// 7.1 Контроль доступа (СКУД)
fbAccessControl(
    VI_System_Time_MS := GVL_STATUS.G_System_Time_MS,
    VI_IsActivePLC := GVL_STATUS.G_Is_Active_PLC,
    VI_Armed := GVL_ALARM.G_Security_Armed,
    VI_System_Mode := GVL_STATE.G_System_Mode,
    VI_Gate_Open_Req := GVL_CONFIG.G_HMI_Gate_Open_Req,
    VI_Wicket_Open_Req := GVL_CONFIG.G_HMI_Wicket_Open_Req,
    VI_Lock_1_Open_Req := GVL_CONFIG.G_HMI_Lock_1_Open_Req,
    VI_Lock_1_Close_Req := GVL_CONFIG.G_HMI_Lock_1_Close_Req,
    VI_Lock_2_Open_Req := GVL_CONFIG.G_HMI_Lock_2_Open_Req,
    VI_Lock_2_Close_Req := GVL_CONFIG.G_HMI_Lock_2_Close_Req,
    VI_PIN_Code := GVL_INTENT_USER.I_PIN_Code,
    VI_RFID_Tag := GVL_INTENT_USER.I_RFID_Tag,
    VI_Access_Codes := GVL_Retain.G_Access_Codes,
    VI_RFID_Tags := GVL_Retain.G_RFID_Tags,
    VI_Config := GVL_CONFIG.G_Security_Config,
    VO_Gate_Open => GVL_INTENT_USER.I_Gate_Open_Request,
    VO_Wicket_Open => GVL_INTENT_USER.I_Wicket_Open_Request,
    VO_Lock_1_Open => GVL_INTENT_USER.I_Lock_1_Open_Request,
    VO_Lock_1_Close => GVL_INTENT_USER.I_Lock_1_Close_Request,
    VO_Lock_2_Open => GVL_INTENT_USER.I_Lock_2_Open_Request,
    VO_Lock_2_Close => GVL_INTENT_USER.I_Lock_2_Close_Request
);
          
END_PROGRAM

PROGRAM PRG_Safety_Operator
  VAR
    fbSafetyWorkflow : FB_Safety_Workflow_Manager;
  END_VAR

            // Operator / test / recover workflow ownership.

fbSafetyWorkflow(
    VI_System_Time_MS := GVL_TIME_SERVICE.G_Now_MS,
    VI_Water_Selective_Recover := GVL_INTENT_USER.I_Water_Selective_Recover,
    VI_Gas_Selective_Recover := GVL_INTENT_USER.I_Gas_Selective_Recover,
    VI_Water_Valve_Test_Open := GVL_INTENT_USER.I_Water_Valve_Test_Open,
    VI_Water_Valve_Test_Close := GVL_INTENT_USER.I_Water_Valve_Test_Close,
    VI_Water_Valve_Test_Confirm := GVL_INTENT_USER.I_Water_Valve_Test_Confirm,
    VI_Gas_Valve_Test_Open := GVL_INTENT_USER.I_Gas_Valve_Test_Open,
    VI_Gas_Valve_Test_Close := GVL_INTENT_USER.I_Gas_Valve_Test_Close,
    VI_Gas_Valve_Test_Confirm := GVL_INTENT_USER.I_Gas_Valve_Test_Confirm
);

// propagate test timeout safety actions
IF fbSafetyWorkflow.VO_Water_Test_Timeout_Close_Required THEN
    GVL_INTENT_SAFETY.I_Test_Timeout_Water_Close := TRUE;
END_IF;

IF fbSafetyWorkflow.VO_Gas_Test_Timeout_Close_Required THEN
    GVL_INTENT_SAFETY.I_Test_Timeout_Gas_Close := TRUE;
END_IF;

// move recovery manual confirm here
IF GVL_INTENT_USER.I_Reset_Errors THEN
    GVL_SAFETY_RECOVERY.G_Recovery_Manual_Confirm := TRUE;
END_IF;

// >>> BULK_SYNC_ANCHOR: PRG_Safety_Operator <<<
          
END_PROGRAM

PROGRAM PRG_System_Runtime_Base
  VAR
    fbSystemInit : FB_System_Init;
    fbSystemRecovery : FB_System_Recovery;
    fbSystemPersist : FB_System_Persist_Manager;
    L_Local_State : ST_System_State_Snapshot;
    L_Remote_State : ST_System_State_Snapshot;
    L_Persist_Buffer : ARRAY[0..4] OF BYTE;
    L_Last_Written_Persist_Buffer : ARRAY[0..4] OF BYTE;
    L_Persist_Buffer_Changed : BOOL;
    L_Last_Persist_Write_MS : UDINT;
    L_Recovery_Done : BOOL;
    L_NVRAM_Cmd : BYTE;
    L_NVRAM_Offset : UDINT;
    L_NVRAM_Done : BOOL;
    L_NVRAM_Err : BOOL;
    L_NVRAM_ErrID : UDINT;
  END_VAR

            // ======================================================
// SYSTEM RUNTIME BASE
// ======================================================
// Initializes and maintains base system runtime helpers.
//
// Legacy direct-state redundancy orchestration is intentionally
// disconnected from active runtime execution.
// Current HA/distributed runtime path is:
// PRG_Peer_Heartbeat_Ingestion -> PRG_Peer_Session_Publication
// -> PRG_HA_Session_Replication -> distributed ingestion/governors.
//
// Do not reconnect FB_System_Redundancy_Orchestrator here without
// explicit barrier/governance review.
// ======================================================

fbSystemInit(
    VIO_Local_State := L_Local_State,
    VIO_Remote_State := L_Remote_State
);

fbSystemRecovery(
    VIO_Recovery_Done := L_Recovery_Done
);

fbSystemPersist(
    VI_System_Time_MS := GVL_TIME_SERVICE.G_Now_MS,
    VI_IsActivePLC := GVL_STATUS.G_Is_Active_PLC,
    VIO_Persist_Buffer := L_Persist_Buffer,
    VIO_Last_Written_Persist_Buffer := L_Last_Written_Persist_Buffer,
    VIO_Persist_Buffer_Changed := L_Persist_Buffer_Changed,
    VIO_Last_Persist_Write_MS := L_Last_Persist_Write_MS,
    VIO_NVRAM_Cmd := L_NVRAM_Cmd,
    VIO_NVRAM_Offset := L_NVRAM_Offset,
    VIO_NVRAM_Done := L_NVRAM_Done,
    VIO_NVRAM_Err := L_NVRAM_Err,
    VIO_NVRAM_ErrID := L_NVRAM_ErrID
);

// >>> BULK_SYNC_ANCHOR: PRG_System_Runtime_Base <<<
          
END_PROGRAM

PROGRAM PRG_Distributed_Snapshot_Governor
  VAR
    L_Now_MS : UDINT;
    L_Delta_MS : UDINT;
    L_Distributed_Snapshot_Valid : BOOL := TRUE;
    L_Error_Code : UDINT := 0;
    L_Error_Text : STRING(160) := '';
    L_Peer_Session_Active : BOOL := FALSE;
  END_VAR

            L_Now_MS := GVL_STATUS.G_System_Time_MS;
L_Distributed_Snapshot_Valid := TRUE;
L_Error_Code := 0;
L_Error_Text := '';

// ======================================================
// DISTRIBUTED IMMUTABLE SNAPSHOT GOVERNOR
// ======================================================
// Governs immutable peer publication snapshot exchange.
// Publication-authoritative only.
// Does not invalidate runtime barrier, PLC fencing
// or local immutable snapshot freeze.
//
// Recovery/release is convergence-lease based:
// distributed snapshot quarantine is not released on a
// single healthy scan.
// ======================================================

GVL_DISTRIBUTED_SNAPSHOT.Peer_Publication_Stale := FALSE;
GVL_DISTRIBUTED_SNAPSHOT.Peer_Snapshot_Not_Immutable := FALSE;
GVL_DISTRIBUTED_SNAPSHOT.Peer_Publication_Divergence := FALSE;
GVL_DISTRIBUTED_SNAPSHOT.Peer_Publication_Reconciliation_Lost := FALSE;
GVL_DISTRIBUTED_SNAPSHOT.Peer_Snapshot_Lease_Expired := FALSE;

// ------------------------------------------------------
// Local immutable publication projection.
// ------------------------------------------------------
// Distributed snapshot is upstream of output freshness in MAIN.
// Therefore local publication baseline must not read GVL_OUTPUT_EPOCH.
// It uses the already-frozen runtime snapshot epoch instead.
// ------------------------------------------------------

GVL_DISTRIBUTED_SNAPSHOT.Local_Distributed_Snapshot_Epoch := GVL_DISTRIBUTED_SNAPSHOT.Distributed_Snapshot_Epoch;
GVL_DISTRIBUTED_SNAPSHOT.Local_Runtime_Snapshot_Epoch := GVL_RUNTIME_SNAPSHOT.Snapshot_Epoch;
GVL_DISTRIBUTED_SNAPSHOT.Local_Publication_Epoch := GVL_RUNTIME_SNAPSHOT.Snapshot_Publication_Epoch;

// ------------------------------------------------------
// Local immutable publication freeze semantics.
// ------------------------------------------------------

IF GVL_RUNTIME_SNAPSHOT.Snapshot_Frozen
AND GVL_RUNTIME_SNAPSHOT.Snapshot_Publication_Allowed
AND GVL_RUNTIME_SNAPSHOT.Snapshot_Copy_Valid
AND GVL_RUNTIME_SNAPSHOT.Snapshot_Isolation_Valid
THEN
    GVL_DISTRIBUTED_SNAPSHOT.Distributed_Snapshot_Frozen := TRUE;
ELSE
    GVL_DISTRIBUTED_SNAPSHOT.Distributed_Snapshot_Frozen := FALSE;

    L_Distributed_Snapshot_Valid := FALSE;
    L_Error_Code := 14000;
    L_Error_Text := 'Local immutable snapshot not frozen';
END_IF;

// ------------------------------------------------------
// Peer session detection.
// ------------------------------------------------------

IF GVL_DISTRIBUTED_SNAPSHOT.Peer_Publication_Epoch > 0 THEN
    L_Peer_Session_Active := TRUE;
END_IF;

IF GVL_DISTRIBUTED_SNAPSHOT.Peer_Runtime_Snapshot_Epoch > 0 THEN
    L_Peer_Session_Active := TRUE;
END_IF;

IF GVL_DISTRIBUTED_SNAPSHOT.Peer_Distributed_Snapshot_Epoch > 0 THEN
    L_Peer_Session_Active := TRUE;
END_IF;

IF GVL_DISTRIBUTED_SNAPSHOT.Peer_Snapshot_Immutable THEN
    L_Peer_Session_Active := TRUE;
END_IF;

// ------------------------------------------------------
// Peer snapshot lease validation.
// ------------------------------------------------------

IF L_Distributed_Snapshot_Valid AND L_Peer_Session_Active THEN
    L_Delta_MS := L_Now_MS - GVL_DISTRIBUTED_SNAPSHOT.Peer_Snapshot_Last_Refresh_MS;

    IF GVL_DISTRIBUTED_SNAPSHOT.Peer_Snapshot_Lease_Active THEN
        IF L_Delta_MS > GVL_DISTRIBUTED_SNAPSHOT.Peer_Snapshot_Lease_Timeout_MS THEN
            GVL_DISTRIBUTED_SNAPSHOT.Peer_Snapshot_Lease_Expired := TRUE;

            L_Distributed_Snapshot_Valid := FALSE;
            L_Error_Code := 14001;
            L_Error_Text := 'Peer snapshot lease expired';
        END_IF;
    END_IF;
END_IF;

// ------------------------------------------------------
// Peer immutable snapshot semantics.
// ------------------------------------------------------

IF L_Distributed_Snapshot_Valid AND L_Peer_Session_Active THEN
    IF NOT GVL_DISTRIBUTED_SNAPSHOT.Peer_Snapshot_Immutable THEN
        GVL_DISTRIBUTED_SNAPSHOT.Peer_Snapshot_Not_Immutable := TRUE;

        L_Distributed_Snapshot_Valid := FALSE;
        L_Error_Code := 14002;
        L_Error_Text := 'Peer snapshot not immutable';
    END_IF;
END_IF;

// ------------------------------------------------------
// Peer publication continuity.
// ------------------------------------------------------

IF L_Distributed_Snapshot_Valid AND L_Peer_Session_Active THEN
    IF GVL_DISTRIBUTED_SNAPSHOT.Peer_Publication_Epoch < GVL_DISTRIBUTED_SNAPSHOT.Local_Publication_Epoch THEN
        GVL_DISTRIBUTED_SNAPSHOT.Peer_Publication_Stale := TRUE;
    END_IF;
END_IF;

// ------------------------------------------------------
// Peer publication reconciliation continuity.
// ------------------------------------------------------

IF L_Distributed_Snapshot_Valid AND L_Peer_Session_Active THEN
    IF GVL_DISTRIBUTED_SNAPSHOT.Peer_Runtime_Snapshot_Epoch <> GVL_DISTRIBUTED_SNAPSHOT.Local_Runtime_Snapshot_Epoch THEN
        GVL_DISTRIBUTED_SNAPSHOT.Peer_Publication_Divergence := TRUE;
    END_IF;
END_IF;

IF GVL_DISTRIBUTED_SNAPSHOT.Peer_Publication_Stale
OR GVL_DISTRIBUTED_SNAPSHOT.Peer_Publication_Divergence
OR GVL_DISTRIBUTED_SNAPSHOT.Peer_Snapshot_Not_Immutable
THEN
    GVL_DISTRIBUTED_SNAPSHOT.Peer_Publication_Reconciliation_Lost := TRUE;
END_IF;

// ------------------------------------------------------
// Publish authoritative distributed snapshot state.
// ------------------------------------------------------

IF L_Distributed_Snapshot_Valid THEN
    GVL_DISTRIBUTED_SNAPSHOT.Distributed_Snapshot_Epoch := GVL_DISTRIBUTED_SNAPSHOT.Distributed_Snapshot_Epoch + 1;
    GVL_DISTRIBUTED_SNAPSHOT.Distributed_Snapshot_Reconciliation_Epoch := GVL_DISTRIBUTED_SNAPSHOT.Distributed_Snapshot_Reconciliation_Epoch + 1;

    GVL_DISTRIBUTED_SNAPSHOT.Distributed_Publication_Reconciled := TRUE;
    GVL_DISTRIBUTED_SNAPSHOT.Distributed_Publication_Freeze_Valid := TRUE;
    GVL_DISTRIBUTED_SNAPSHOT.Distributed_Snapshot_Consistent := TRUE;

    // Lease-based recovery release.
    IF GVL_CONVERGENCE.Convergence_Release_Allowed THEN
        GVL_DISTRIBUTED_SNAPSHOT.Distributed_Snapshot_Quarantine_Active := FALSE;
    END_IF;

    GVL_DISTRIBUTED_SNAPSHOT.Distributed_Snapshot_Last_Error_Code := 0;
    GVL_DISTRIBUTED_SNAPSHOT.Distributed_Snapshot_Last_Error_Text := '';
ELSE
    // Invalid distributed snapshot state escalates immediately.
    GVL_DISTRIBUTED_SNAPSHOT.Distributed_Publication_Reconciled := FALSE;
    GVL_DISTRIBUTED_SNAPSHOT.Distributed_Publication_Freeze_Valid := FALSE;
    GVL_DISTRIBUTED_SNAPSHOT.Distributed_Snapshot_Consistent := FALSE;

    GVL_DISTRIBUTED_SNAPSHOT.Distributed_Snapshot_Quarantine_Active := TRUE;

    GVL_DISTRIBUTED_SNAPSHOT.Distributed_Snapshot_Last_Error_Code := L_Error_Code;
    GVL_DISTRIBUTED_SNAPSHOT.Distributed_Snapshot_Last_Error_Text := L_Error_Text;
END_IF;
          
END_PROGRAM

PROGRAM PRG_Semantic_Federation_Governor
  VAR
    L_Now_MS : UDINT;
    L_Federation_Valid : BOOL := TRUE;
    L_Error_Code : UDINT := 0;
    L_Error_Text : STRING(160) := '';
  END_VAR

            L_Now_MS := GVL_STATUS.G_System_Time_MS;
L_Federation_Valid := TRUE;
L_Error_Code := 0;
L_Error_Text := '';

// Fail-safe defaults.
GVL_SEMANTIC_FEDERATION_FABRIC.Semantic_Federation_Valid := FALSE;
GVL_SEMANTIC_FEDERATION_FABRIC.Semantic_Federation_Granted := FALSE;
GVL_SEMANTIC_FEDERATION_FABRIC.Semantic_Federation_Quarantine_Active := TRUE;

GVL_SEMANTIC_FEDERATION_FABRIC.External_SCADA_Semantics_Coherent := FALSE;
GVL_SEMANTIC_FEDERATION_FABRIC.Cloud_Authority_Projection_Aligned := FALSE;
GVL_SEMANTIC_FEDERATION_FABRIC.MQTT_Semantic_State_Fresh := FALSE;
GVL_SEMANTIC_FEDERATION_FABRIC.ThirdParty_Integration_Trust_Valid := FALSE;
GVL_SEMANTIC_FEDERATION_FABRIC.Federated_Observability_Coherent := FALSE;

// Operator semantic alignment required.
IF NOT GVL_OPERATOR_SEMANTIC_ALIGNMENT.Operator_Semantic_Alignment_Granted THEN
    L_Federation_Valid := FALSE;
    L_Error_Code := 41000;
    L_Error_Text := 'Operator semantic alignment not granted';
END_IF;

// Ecosystem semantic split-brain detectors.
IF GVL_SEMANTIC_FEDERATION_FABRIC.External_Semantic_Lag_Detected THEN
    L_Federation_Valid := FALSE;
    L_Error_Code := 41001;
    L_Error_Text := 'External semantic lag detected';
END_IF;

IF GVL_SEMANTIC_FEDERATION_FABRIC.SCADA_Projection_Skew_Detected THEN
    L_Federation_Valid := FALSE;
    L_Error_Code := 41002;
    L_Error_Text := 'SCADA projection skew detected';
END_IF;

IF GVL_SEMANTIC_FEDERATION_FABRIC.Cloud_Authority_Desynchronization_Detected THEN
    L_Federation_Valid := FALSE;
    L_Error_Code := 41003;
    L_Error_Text := 'Cloud authority desynchronization detected';
END_IF;

IF GVL_SEMANTIC_FEDERATION_FABRIC.ThirdParty_Semantic_Drift_Detected THEN
    L_Federation_Valid := FALSE;
    L_Error_Code := 41004;
    L_Error_Text := 'Third-party semantic drift detected';
END_IF;

IF GVL_SEMANTIC_FEDERATION_FABRIC.Integration_Trust_Divergence_Detected THEN
    L_Federation_Valid := FALSE;
    L_Error_Code := 41005;
    L_Error_Text := 'Integration trust divergence detected';
END_IF;

IF GVL_SEMANTIC_FEDERATION_FABRIC.Federated_Authority_Inconsistency_Detected THEN
    L_Federation_Valid := FALSE;
    L_Error_Code := 41006;
    L_Error_Text := 'Federated authority inconsistency detected';
END_IF;

// External semantic federation validation.
IF L_Federation_Valid
AND NOT GVL_SEMANTIC_FEDERATION_FABRIC.Exported_Authority_State_Coherent THEN
    L_Federation_Valid := FALSE;
    L_Error_Code := 41010;
    L_Error_Text := 'Exported authority state coherence invalid';
END_IF;

IF L_Federation_Valid
AND NOT GVL_SEMANTIC_FEDERATION_FABRIC.Federation_Projection_Temporal_Stable THEN
    L_Federation_Valid := FALSE;
    L_Error_Code := 41011;
    L_Error_Text := 'Federation projection temporal stability invalid';
END_IF;

IF L_Federation_Valid
AND NOT GVL_SEMANTIC_FEDERATION_FABRIC.External_Runtime_Interpretation_Aligned THEN
    L_Federation_Valid := FALSE;
    L_Error_Code := 41012;
    L_Error_Text := 'External runtime interpretation alignment invalid';
END_IF;

IF L_Federation_Valid
AND NOT GVL_SEMANTIC_FEDERATION_FABRIC.Federated_Trust_Boundary_Stable THEN
    L_Federation_Valid := FALSE;
    L_Error_Code := 41013;
    L_Error_Text := 'Federated trust boundary unstable';
END_IF;

IF L_Federation_Valid THEN
    GVL_SEMANTIC_FEDERATION_FABRIC.Semantic_Federation_Valid := TRUE;
    GVL_SEMANTIC_FEDERATION_FABRIC.Semantic_Federation_Granted := TRUE;
    GVL_SEMANTIC_FEDERATION_FABRIC.Semantic_Federation_Quarantine_Active := FALSE;

    GVL_SEMANTIC_FEDERATION_FABRIC.External_SCADA_Semantics_Coherent := TRUE;
    GVL_SEMANTIC_FEDERATION_FABRIC.Cloud_Authority_Projection_Aligned := TRUE;
    GVL_SEMANTIC_FEDERATION_FABRIC.MQTT_Semantic_State_Fresh := TRUE;
    GVL_SEMANTIC_FEDERATION_FABRIC.ThirdParty_Integration_Trust_Valid := TRUE;
    GVL_SEMANTIC_FEDERATION_FABRIC.Federated_Observability_Coherent := TRUE;

    GVL_SEMANTIC_FEDERATION_FABRIC.Semantic_Federation_Epoch :=
        GVL_OPERATOR_SEMANTIC_ALIGNMENT.Operator_Alignment_Epoch;

    GVL_SEMANTIC_FEDERATION_FABRIC.Semantic_Federation_Epoch_Coherent := TRUE;

    GVL_SEMANTIC_FEDERATION_FABRIC.Semantic_Federation_Last_Update_MS :=
        L_Now_MS;

    GVL_SEMANTIC_FEDERATION_FABRIC.Semantic_Federation_Lease_Expired := FALSE;

    GVL_SEMANTIC_FEDERATION_FABRIC.Semantic_Federation_Last_Error_Code := 0;
    GVL_SEMANTIC_FEDERATION_FABRIC.Semantic_Federation_Last_Error_Text := '';
ELSE
    GVL_SEMANTIC_FEDERATION_FABRIC.Semantic_Federation_Valid := FALSE;
    GVL_SEMANTIC_FEDERATION_FABRIC.Semantic_Federation_Granted := FALSE;
    GVL_SEMANTIC_FEDERATION_FABRIC.Semantic_Federation_Quarantine_Active := TRUE;

    GVL_SEMANTIC_FEDERATION_FABRIC.Semantic_Federation_Lease_Expired := TRUE;

    GVL_SEMANTIC_FEDERATION_FABRIC.Semantic_Federation_Last_Error_Code :=
        L_Error_Code;

    GVL_SEMANTIC_FEDERATION_FABRIC.Semantic_Federation_Last_Error_Text :=
        L_Error_Text;

    GVL_SEMANTIC_FEDERATION_FABRIC.Semantic_Federation_Invalidation_Count :=
        GVL_SEMANTIC_FEDERATION_FABRIC.Semantic_Federation_Invalidation_Count + 1;
END_IF;
          
END_PROGRAM

PROGRAM PRG_Survivability_Intelligence_Governor

            // ADVISORY SURVIVABILITY INTELLIGENCE
// READ-ONLY / NON-INVASIVE
// NO ACTUATION / AUTHORITY / RECOVERY MUTATION

GVL_SURVIVABILITY_INTELLIGENCE_FABRIC.System_Survivable :=
    GVL_PHYSICAL_REALITY_VERIFICATION_FABRIC.Physical_Runtime_Reality_Valid;

GVL_SURVIVABILITY_INTELLIGENCE_FABRIC.Degraded_But_Safe :=
    GVL_RUNTIME_STATE_ALGEBRA.Current_Runtime_State = SYS_DEGRADED;

GVL_SURVIVABILITY_INTELLIGENCE_FABRIC.Isolated_But_Stable :=
    GVL_RUNTIME_STATE_ALGEBRA.Current_Runtime_State = SYS_ISOLATED;

GVL_SURVIVABILITY_INTELLIGENCE_FABRIC.Partitioned_But_Survivable :=
    GVL_RUNTIME_STATE_ALGEBRA.Current_Runtime_State = SYS_PARTITIONED;

GVL_SURVIVABILITY_INTELLIGENCE_FABRIC.Resource_Starved_But_Recoverable :=
    GVL_OPERATIONAL_INTELLIGENCE_FABRIC.Governance_Complexity_Pressure_Observed;

GVL_SURVIVABILITY_INTELLIGENCE_FABRIC.Essential_Functions_Preserved :=
    GVL_SAFETY_OBSERVABILITY_TRUTH_FABRIC.Observability_Reality_Equivalence_Granted;

IF GVL_OPERATIONAL_INTELLIGENCE_FABRIC.Governance_Saturation_Observed THEN
    GVL_SURVIVABILITY_INTELLIGENCE_FABRIC.NonEssential_Shedding_Recommended := TRUE;
    GVL_SURVIVABILITY_INTELLIGENCE_FABRIC.Heavy_Diagnostics_Defer_Recommended := TRUE;
    GVL_SURVIVABILITY_INTELLIGENCE_FABRIC.Trend_Analytics_Defer_Recommended := TRUE;
END_IF;

IF GVL_OPERATIONAL_INTELLIGENCE_FABRIC.Governance_Complexity_Pressure_Observed THEN
    GVL_SURVIVABILITY_INTELLIGENCE_FABRIC.Telemetry_Rate_Reduction_Recommended := TRUE;
END_IF;

IF GVL_RUNTIME_TRANSITION_SYSTEM.Illegal_Runtime_Transition_Observed THEN
    GVL_SURVIVABILITY_INTELLIGENCE_FABRIC.LongDuration_Degradation_Observed := TRUE;
    GVL_SURVIVABILITY_INTELLIGENCE_FABRIC.Chronic_Degradation_Risk_Increasing := TRUE;
    GVL_SURVIVABILITY_INTELLIGENCE_FABRIC.Survivability_Advisory_Available := TRUE;
    GVL_SURVIVABILITY_INTELLIGENCE_FABRIC.Survivability_Advisory_Code :=
        'survivability degraded under prolonged instability';
END_IF;

GVL_SURVIVABILITY_INTELLIGENCE_FABRIC.Governance_Saturation_Pressure_Observed :=
    GVL_OPERATIONAL_INTELLIGENCE_FABRIC.Governance_Saturation_Observed;

GVL_SURVIVABILITY_INTELLIGENCE_FABRIC.Distributed_Instability_Pressure_Observed :=
    NOT GVL_DISTRIBUTED_SAFETY_REALITY_CONSENSUS_FABRIC.Distributed_Safety_Consensus_Valid;
          
END_PROGRAM

PROGRAM PRG_Authority_Restoration_Governor
  VAR
    L_Now_MS : UDINT;
    L_Restoration_Valid : BOOL := TRUE;
  END_VAR

            L_Now_MS := GVL_STATUS.G_System_Time_MS;
L_Restoration_Valid := TRUE;

// Fail-safe defaults.
GVL_AUTHORITY_RESTORATION.Authority_Restoration_Active := FALSE;
GVL_AUTHORITY_RESTORATION.Authority_Restoration_Allowed := FALSE;
GVL_AUTHORITY_RESTORATION.Authority_Restoration_Completed := FALSE;

GVL_AUTHORITY_RESTORATION.Snapshot_Restoration_Valid := FALSE;
GVL_AUTHORITY_RESTORATION.Consensus_Restoration_Valid := FALSE;
GVL_AUTHORITY_RESTORATION.Causality_Restoration_Valid := FALSE;
GVL_AUTHORITY_RESTORATION.Epoch_Restoration_Valid := FALSE;
GVL_AUTHORITY_RESTORATION.Lineage_Restoration_Valid := FALSE;

GVL_AUTHORITY_RESTORATION.Revocation_Clearance_Valid := FALSE;
GVL_AUTHORITY_RESTORATION.Stabilization_Window_Elapsed := FALSE;
GVL_AUTHORITY_RESTORATION.Reauthorization_Order_Valid := FALSE;

// Restoration impossible while revocation active.
IF GVL_AUTHORITY_REVOCATION.Authority_Revocation_Active THEN
    L_Restoration_Valid := FALSE;
END_IF;

// Snapshot must recover first.
IF L_Restoration_Valid
AND NOT GVL_PHYSICAL_SNAPSHOT.Physical_Snapshot_Valid THEN
    L_Restoration_Valid := FALSE;
END_IF;

IF L_Restoration_Valid THEN
    GVL_AUTHORITY_RESTORATION.Snapshot_Restoration_Valid := TRUE;
END_IF;

// Consensus recovery.
IF L_Restoration_Valid
AND NOT GVL_SENSOR_CONSENSUS.Sensor_Consensus_Valid THEN
    L_Restoration_Valid := FALSE;
END_IF;

IF L_Restoration_Valid THEN
    GVL_AUTHORITY_RESTORATION.Consensus_Restoration_Valid := TRUE;
END_IF;

// Telemetry causality recovery.
IF L_Restoration_Valid
AND NOT GVL_TELEMETRY.Command_Telemetry_Causality_Valid THEN
    L_Restoration_Valid := FALSE;
END_IF;

IF L_Restoration_Valid THEN
    GVL_AUTHORITY_RESTORATION.Causality_Restoration_Valid := TRUE;
END_IF;

// Epoch coherence recovery.
IF L_Restoration_Valid
AND NOT GVL_PHYSICAL_AUTHORITY_EPOCH.Physical_Authority_Epoch_Valid THEN
    L_Restoration_Valid := FALSE;
END_IF;

IF L_Restoration_Valid THEN
    GVL_AUTHORITY_RESTORATION.Epoch_Restoration_Valid := TRUE;
END_IF;

// Lineage continuity recovery.
IF L_Restoration_Valid
AND NOT GVL_AUTHORITY_LINEAGE.Authority_Lineage_Valid THEN
    L_Restoration_Valid := FALSE;
END_IF;

IF L_Restoration_Valid THEN
    GVL_AUTHORITY_RESTORATION.Lineage_Restoration_Valid := TRUE;
END_IF;

// Revocation must be fully cleared.
IF L_Restoration_Valid
AND GVL_AUTHORITY_REVOCATION.Quarantine_Fabric_Active THEN
    L_Restoration_Valid := FALSE;
END_IF;

IF L_Restoration_Valid THEN
    GVL_AUTHORITY_RESTORATION.Revocation_Clearance_Valid := TRUE;
END_IF;

// Stabilization window after recovery.
IF L_Restoration_Valid
AND ((L_Now_MS - GVL_AUTHORITY_REVOCATION.Revocation_Last_Update_MS) < 5000) THEN
    L_Restoration_Valid := FALSE;
END_IF;

IF L_Restoration_Valid THEN
    GVL_AUTHORITY_RESTORATION.Stabilization_Window_Elapsed := TRUE;
END_IF;

IF L_Restoration_Valid THEN
    GVL_AUTHORITY_RESTORATION.Authority_Restoration_Active := TRUE;
    GVL_AUTHORITY_RESTORATION.Authority_Restoration_Allowed := TRUE;
    GVL_AUTHORITY_RESTORATION.Authority_Restoration_Completed := TRUE;

    GVL_AUTHORITY_RESTORATION.Reauthorization_Order_Valid := TRUE;

    GVL_AUTHORITY_RESTORATION.Restoration_Epoch :=
        GVL_PHYSICAL_AUTHORITY_EPOCH.Physical_Authority_Epoch;

    GVL_AUTHORITY_RESTORATION.Restoration_Last_Update_MS := L_Now_MS;
END_IF;
          
END_PROGRAM

PROGRAM PRG_System_Simulation
  VAR
    fbSimulation : FB_Simulation_Manager;
    fbPlayback : FB_Presence_Playback;
    L_Playback_Lights : ARRAY[1..32] OF BOOL;
    L_Scenario_Config : ST_Scenario_Config;
  END_VAR

            L_Scenario_Config := GVL_CONFIG.G_HMI_Scenario_Configs[TO_INT(GVL_STATUS.G_Current_Scenario)];

fbSimulation(
    VI_System_Time_MS := GVL_TIME_SERVICE.G_Now_MS,
    VI_IsActivePLC := GVL_STATUS.G_Is_Active_PLC,
    VI_Scenario := GVL_STATUS.G_Current_Scenario,
    VI_Config := L_Scenario_Config
);

fbPlayback(
    VI_Mode_Record := FALSE,
    VI_Time_Index := GVL_TIME_SERVICE.G_Now_MS,
    VI_Light_Inputs := L_Playback_Lights
);

// Reset outputs
GVL_SIMULATION.G_Sim_Heating_Sensor_Fault := FALSE;
GVL_SIMULATION.G_Sim_IO_Fault := FALSE;
GVL_SIMULATION.G_Sim_Low_Pressure := FALSE;
GVL_SIMULATION.G_Sim_Predictive_Pump_Fault := FALSE;
GVL_SIMULATION.G_Sim_Gas_Alarm := FALSE;
GVL_SIMULATION.G_Sim_Leak_Alarm := FALSE;
GVL_SIMULATION.G_Sim_Smoke_Alarm := FALSE;
GVL_SIMULATION.G_Sim_Dual_PLC_Active := FALSE;

IF NOT GVL_SIMULATION.G_Simulation_Enable THEN
    GVL_SIMULATION.G_Test_Running := FALSE;
    GVL_SIMULATION.G_Test_Scenario_Active := FALSE;
    RETURN;
END_IF;

// Start scenario
IF GVL_SIMULATION.G_Test_Start THEN
    GVL_SIMULATION.G_Test_Scenario_Active := TRUE;
    GVL_SIMULATION.G_Test_Started_MS := GVL_TIME_SERVICE.G_Now_MS;
END_IF;

// Stop scenario
IF GVL_SIMULATION.G_Test_Stop THEN
    GVL_SIMULATION.G_Test_Scenario_Active := FALSE;
END_IF;

GVL_SIMULATION.G_Test_Running := GVL_SIMULATION.G_Test_Scenario_Active;

IF NOT GVL_SIMULATION.G_Test_Scenario_Active THEN
    RETURN;
END_IF;

// Scenario execution
CASE GVL_SIMULATION.G_Test_Scenario_ID OF

    1: // Gas safety
        GVL_SIMULATION.G_Sim_Gas_Alarm := TRUE;
        GVL_SIMULATION.G_Test_Expected_Result_Code := 1;

    2: // Leak + pressure
        GVL_SIMULATION.G_Sim_Leak_Alarm := TRUE;
        GVL_SIMULATION.G_Sim_Low_Pressure := TRUE;
        GVL_SIMULATION.G_Test_Expected_Result_Code := 2;

    3: // Sensor + predictive
        GVL_SIMULATION.G_Sim_Heating_Sensor_Fault := TRUE;
        GVL_SIMULATION.G_Sim_Predictive_Pump_Fault := TRUE;
        GVL_SIMULATION.G_Test_Expected_Result_Code := 2;

    4: // Dual PLC
        GVL_SIMULATION.G_Sim_Dual_PLC_Active := TRUE;
        GVL_SIMULATION.G_Test_Expected_Result_Code := 3;

    5: // Full stress
        GVL_SIMULATION.G_Sim_Gas_Alarm := TRUE;
        GVL_SIMULATION.G_Sim_Leak_Alarm := TRUE;
        GVL_SIMULATION.G_Sim_Smoke_Alarm := TRUE;
        GVL_SIMULATION.G_Sim_Low_Pressure := TRUE;
        GVL_SIMULATION.G_Sim_Predictive_Pump_Fault := TRUE;
        GVL_SIMULATION.G_Test_Expected_Result_Code := 4;

ELSE
        // No fallback required
END_CASE;

// Auto stop by time
IF (GVL_TIME_SERVICE.G_Now_MS - GVL_SIMULATION.G_Test_Started_MS) > GVL_SIMULATION.G_Test_Duration_MS THEN
    GVL_SIMULATION.G_Test_Scenario_Active := FALSE;
END_IF;

// >>> BULK_SYNC_ANCHOR: PRG_System_Simulation <<<
          
END_PROGRAM

PROGRAM PRG_Distributed_Snapshot_Publication

            // ======================================================
// DISTRIBUTED SNAPSHOT PUBLICATION
// ======================================================
// Canonical local distributed snapshot export into the
// HA replication boundary.
//
// Purpose:
// publish normalized immutable snapshot/publication state
// into the dedicated HA boundary before snapshot ingestion.
//
// This layer does NOT:
// - perform reconciliation
// - validate peer snapshot state
// - arbitrate distributed publication authority
//
// Disabled HA replication must not leave stale snapshot mirrors.
// ======================================================

IF NOT GVL_HA_SESSION_REPLICATION.HA_Replication_Enabled THEN
    GVL_HA_SESSION_REPLICATION.HA_Remote_Distributed_Snapshot_Epoch := 0;
    GVL_HA_SESSION_REPLICATION.HA_Remote_Runtime_Snapshot_Epoch := 0;
    GVL_HA_SESSION_REPLICATION.HA_Remote_Publication_Epoch := 0;
    GVL_HA_SESSION_REPLICATION.HA_Remote_Snapshot_Immutable := FALSE;
    GVL_HA_SESSION_REPLICATION.HA_Remote_Snapshot_Last_Refresh_MS := 0;
    RETURN;
END_IF;

GVL_HA_SESSION_REPLICATION.HA_Remote_Distributed_Snapshot_Epoch :=
    GVL_DISTRIBUTED_SNAPSHOT.Local_Distributed_Snapshot_Epoch;

GVL_HA_SESSION_REPLICATION.HA_Remote_Runtime_Snapshot_Epoch :=
    GVL_RUNTIME_SNAPSHOT.Snapshot_Epoch;

GVL_HA_SESSION_REPLICATION.HA_Remote_Publication_Epoch :=
    GVL_RUNTIME_SNAPSHOT.Snapshot_Publication_Epoch;

GVL_HA_SESSION_REPLICATION.HA_Remote_Snapshot_Immutable :=
    GVL_RUNTIME_SNAPSHOT.Snapshot_Frozen
    AND GVL_RUNTIME_SNAPSHOT.Snapshot_Publication_Allowed
    AND GVL_RUNTIME_SNAPSHOT.Snapshot_Copy_Valid
    AND GVL_RUNTIME_SNAPSHOT.Snapshot_Isolation_Valid;

GVL_HA_SESSION_REPLICATION.HA_Remote_Snapshot_Last_Refresh_MS :=
    GVL_STATUS.G_System_Time_MS;

// >>> BULK_SYNC_ANCHOR: PRG_Distributed_Snapshot_Publication <<<
          
END_PROGRAM

PROGRAM PRG_Distributed_Commit_Publication

            // ======================================================
// DISTRIBUTED COMMIT PUBLICATION
// ======================================================
// Canonical local distributed commit export into the
// HA replication boundary.
//
// Purpose:
// publish normalized deterministic commit handshake state
// into the dedicated HA boundary before commit ingestion.
//
// This layer does NOT:
// - perform reconciliation
// - validate peer acknowledgements
// - arbitrate publication authority
//
// Disabled HA replication must not leave stale commit mirrors.
// ======================================================

IF NOT GVL_HA_SESSION_REPLICATION.HA_Replication_Enabled THEN
    GVL_HA_SESSION_REPLICATION.HA_Remote_Publication_Commit_Epoch := 0;
    GVL_HA_SESSION_REPLICATION.HA_Remote_Prepare_Epoch := 0;
    GVL_HA_SESSION_REPLICATION.HA_Remote_Commit_Ack_Valid := FALSE;
    GVL_HA_SESSION_REPLICATION.HA_Remote_Commit_Last_Refresh_MS := 0;
    RETURN;
END_IF;

GVL_HA_SESSION_REPLICATION.HA_Remote_Publication_Commit_Epoch :=
    GVL_DISTRIBUTED_COMMIT.Local_Publication_Commit_Epoch;

GVL_HA_SESSION_REPLICATION.HA_Remote_Prepare_Epoch :=
    GVL_DISTRIBUTED_COMMIT.Local_Prepare_Epoch;

GVL_HA_SESSION_REPLICATION.HA_Remote_Commit_Ack_Valid :=
    GVL_DISTRIBUTED_COMMIT.Publication_Commit_Confirmed;

GVL_HA_SESSION_REPLICATION.HA_Remote_Commit_Last_Refresh_MS :=
    GVL_STATUS.G_System_Time_MS;

// >>> BULK_SYNC_ANCHOR: PRG_Distributed_Commit_Publication <<<
          
END_PROGRAM

PROGRAM PRG_Energy_Resurrection_Boundary_Governor

            IF GVL_POWER_DOMAIN_SEGMENTATION_FABRIC.Power_Domain_Segmentation_Granted
AND NOT GVL_ENERGY_RESURRECTION_BOUNDARY_FABRIC.Unsafe_Energy_Resurrection_Detected
AND NOT GVL_ENERGY_RESURRECTION_BOUNDARY_FABRIC.CrossDomain_Energy_Recovery_Race
AND NOT GVL_ENERGY_RESURRECTION_BOUNDARY_FABRIC.Energy_Recovery_Fork_Detected THEN

    GVL_ENERGY_RESURRECTION_BOUNDARY_FABRIC.Energy_Resurrection_Boundary_Valid := TRUE;
    GVL_ENERGY_RESURRECTION_BOUNDARY_FABRIC.Energy_Resurrection_Boundary_Granted := TRUE;
    GVL_ENERGY_RESURRECTION_BOUNDARY_FABRIC.Energy_Resurrection_Causality_Valid := TRUE;
    GVL_ENERGY_RESURRECTION_BOUNDARY_FABRIC.Energy_Authority_Recovery_Bounded := TRUE;
    GVL_ENERGY_RESURRECTION_BOUNDARY_FABRIC.CrossDomain_Energy_Recovery_Stable := TRUE;
END_IF;
          
END_PROGRAM

PROGRAM PRG_Semantic_Progress_Governor
  VAR
    L_Now_MS : UDINT;
    L_Delta_MS : UDINT;
    L_Semantic_Valid : BOOL := TRUE;
    L_Error_Code : UDINT := 0;
    L_Error_Text : STRING(160) := '';
    L_Runtime_Epoch_Advanced : BOOL := FALSE;
    L_Snapshot_Epoch_Advanced : BOOL := FALSE;
    L_Distributed_Commit_Epoch_Advanced : BOOL := FALSE;
    L_Output_Epoch_Advanced : BOOL := FALSE;
    L_Runtime_Snapshot_Skew : UDINT;
    L_Runtime_Commit_Skew : UDINT;
    L_Runtime_Output_Skew : UDINT;
  END_VAR

            L_Now_MS := GVL_STATUS.G_System_Time_MS;
L_Semantic_Valid := TRUE;
L_Error_Code := 0;
L_Error_Text := '';

GVL_SEMANTIC_PROGRESS.Semantic_Stagnation_Detected := FALSE;
GVL_SEMANTIC_PROGRESS.Semantic_Replay_Suspected := FALSE;
GVL_SEMANTIC_PROGRESS.Semantic_Livelock_Suspected := FALSE;
GVL_SEMANTIC_PROGRESS.Semantic_Deadlock_Suspected := FALSE;
GVL_SEMANTIC_PROGRESS.Semantic_Progress_Lease_Expired := FALSE;
GVL_SEMANTIC_PROGRESS.Semantic_Phase_Stall_Detected := FALSE;
GVL_SEMANTIC_PROGRESS.Semantic_Output_Stall_Detected := FALSE;

GVL_SEMANTIC_PROGRESS.Semantic_Runtime_Barrier_Epoch := ULINT_TO_UDINT(GVL_RUNTIME_EPOCH.Runtime_Epoch);
GVL_SEMANTIC_PROGRESS.Semantic_Runtime_Snapshot_Epoch := ULINT_TO_UDINT(GVL_RUNTIME_SNAPSHOT.Snapshot_Epoch);
GVL_SEMANTIC_PROGRESS.Semantic_Distributed_Commit_Epoch := ULINT_TO_UDINT(GVL_DISTRIBUTED_COMMIT.Distributed_Commit_Epoch);
GVL_SEMANTIC_PROGRESS.Semantic_Output_Publication_Epoch := ULINT_TO_UDINT(GVL_OUTPUT_EPOCH.Output_Publication_Epoch);

GVL_SEMANTIC_PROGRESS.Semantic_Runtime_Barrier_Evidence_OK :=
    GVL_RUNTIME_EPOCH.Runtime_Runtime_Barrier_OK AND
    GVL_RUNTIME_EPOCH.Runtime_Snapshot_Published AND
    GVL_RUNTIME_EPOCH.Runtime_IO_Publication_Allowed;

GVL_SEMANTIC_PROGRESS.Semantic_Runtime_Snapshot_Evidence_OK :=
    GVL_RUNTIME_SNAPSHOT.Snapshot_Frozen AND
    GVL_RUNTIME_SNAPSHOT.Snapshot_Publication_Allowed AND
    GVL_RUNTIME_SNAPSHOT.Snapshot_Copy_Valid AND
    GVL_RUNTIME_SNAPSHOT.Snapshot_Isolation_Valid AND
    GVL_RUNTIME_SNAPSHOT.Snapshot_Runtime_Authority_Valid AND
    NOT GVL_RUNTIME_SNAPSHOT.Snapshot_Mutation_Detected;

GVL_SEMANTIC_PROGRESS.Semantic_Distributed_Commit_Evidence_OK :=
    GVL_DISTRIBUTED_COMMIT.Distributed_Commit_Valid AND
    GVL_DISTRIBUTED_COMMIT.Publication_Prepare_Valid AND
    GVL_DISTRIBUTED_COMMIT.Publication_Commit_Confirmed AND
    NOT GVL_DISTRIBUTED_COMMIT.Peer_Commit_Mismatch AND
    NOT GVL_DISTRIBUTED_COMMIT.Distributed_Commit_Quarantine_Active AND
    NOT GVL_DISTRIBUTED_COMMIT.Commit_Lease_Expired;

GVL_SEMANTIC_PROGRESS.Semantic_Output_Publication_Evidence_OK :=
    GVL_OUTPUT_EPOCH.Output_Publication_Valid AND
    GVL_OUTPUT_EPOCH.Output_Runtime_Epoch_Valid AND
    NOT GVL_OUTPUT_EPOCH.Output_Lease_Expired AND
    NOT GVL_OUTPUT_EPOCH.Output_Stale_Detected AND
    NOT GVL_OUTPUT_EPOCH.Output_Forced_Safe_Decay;
          
END_PROGRAM

PROGRAM PRG_Distributed_Commit_Observability

            // ======================================================
// DISTRIBUTED COMMIT OBSERVABILITY GOVERNOR
// ======================================================
// Isolated downstream observability projection layer.
// Publication visibility only.
// Does not invalidate runtime barrier,
// PLC fencing, immutable snapshots or IO directly.
//
// Visibility ownership rule:
// this layer publishes only dedicated distributed
// visibility fields.
//
// Global observability escalation ownership remains
// inside PRG_Observability_Governor.
// ======================================================

GVL_OBSERVABILITY_AUTHORITY.Distributed_Commit_Visible := FALSE;
GVL_OBSERVABILITY_AUTHORITY.Distributed_Commit_Quarantine_Visible := FALSE;

GVL_OBSERVABILITY_AUTHORITY.Publication_Prepare_Visible := FALSE;
GVL_OBSERVABILITY_AUTHORITY.Publication_Commit_Visible := FALSE;

GVL_OBSERVABILITY_AUTHORITY.Peer_Commit_Ack_Visible := FALSE;
GVL_OBSERVABILITY_AUTHORITY.Peer_Commit_Mismatch_Visible := FALSE;
GVL_OBSERVABILITY_AUTHORITY.Peer_Commit_Replay_Visible := FALSE;
GVL_OBSERVABILITY_AUTHORITY.Peer_Commit_Missing_Visible := FALSE;

GVL_OBSERVABILITY_AUTHORITY.Commit_Lease_Expired_Visible := FALSE;

// ------------------------------------------------------
// Distributed commit validity visibility.
// ------------------------------------------------------

IF NOT GVL_DISTRIBUTED_COMMIT.Distributed_Commit_Valid THEN
    GVL_OBSERVABILITY_AUTHORITY.Distributed_Commit_Visible := TRUE;
END_IF;

IF GVL_DISTRIBUTED_COMMIT.Distributed_Commit_Quarantine_Active THEN
    GVL_OBSERVABILITY_AUTHORITY.Distributed_Commit_Quarantine_Visible := TRUE;
END_IF;

// ------------------------------------------------------
// Publication lifecycle visibility.
// ------------------------------------------------------

IF GVL_DISTRIBUTED_COMMIT.Publication_Prepare_Active THEN
    GVL_OBSERVABILITY_AUTHORITY.Publication_Prepare_Visible := TRUE;
END_IF;

IF GVL_DISTRIBUTED_COMMIT.Publication_Commit_Confirmed THEN
    GVL_OBSERVABILITY_AUTHORITY.Publication_Commit_Visible := TRUE;
END_IF;

// ------------------------------------------------------
// Peer commit continuity visibility.
// ------------------------------------------------------

IF GVL_DISTRIBUTED_COMMIT.Peer_Commit_Ack_Valid THEN
    GVL_OBSERVABILITY_AUTHORITY.Peer_Commit_Ack_Visible := TRUE;
END_IF;

IF GVL_DISTRIBUTED_COMMIT.Peer_Commit_Mismatch THEN
    GVL_OBSERVABILITY_AUTHORITY.Peer_Commit_Mismatch_Visible := TRUE;
END_IF;

IF GVL_DISTRIBUTED_COMMIT.Peer_Commit_Replay_Detected THEN
    GVL_OBSERVABILITY_AUTHORITY.Peer_Commit_Replay_Visible := TRUE;
END_IF;

IF GVL_DISTRIBUTED_COMMIT.Peer_Commit_Missing THEN
    GVL_OBSERVABILITY_AUTHORITY.Peer_Commit_Missing_Visible := TRUE;
END_IF;

IF GVL_DISTRIBUTED_COMMIT.Commit_Lease_Expired THEN
    GVL_OBSERVABILITY_AUTHORITY.Commit_Lease_Expired_Visible := TRUE;
END_IF;
          
END_PROGRAM

PROGRAM PRG_Physical_Deadlock_Resolution_Governor

            IF GVL_ENERGY_RESURRECTION_BOUNDARY_FABRIC.Energy_Resurrection_Boundary_Granted
AND NOT GVL_PHYSICAL_DEADLOCK_RESOLUTION_FABRIC.Physical_CircularWait_Detected
AND NOT GVL_PHYSICAL_DEADLOCK_RESOLUTION_FABRIC.CrossDomain_Progress_Deadlock
AND NOT GVL_PHYSICAL_DEADLOCK_RESOLUTION_FABRIC.Recovery_Livelock_Detected
AND NOT GVL_PHYSICAL_DEADLOCK_RESOLUTION_FABRIC.Physical_Progress_Stall_Detected THEN

    GVL_PHYSICAL_DEADLOCK_RESOLUTION_FABRIC.Physical_Deadlock_Resolution_Valid := TRUE;
    GVL_PHYSICAL_DEADLOCK_RESOLUTION_FABRIC.Physical_Deadlock_Resolution_Granted := TRUE;
    GVL_PHYSICAL_DEADLOCK_RESOLUTION_FABRIC.Deadlock_Resolution_Canonical := TRUE;
    GVL_PHYSICAL_DEADLOCK_RESOLUTION_FABRIC.Physical_Forward_Progress_Valid := TRUE;
    GVL_PHYSICAL_DEADLOCK_RESOLUTION_FABRIC.CrossDomain_Execution_Progress_Stable := TRUE;
END_IF;
          
END_PROGRAM

PROGRAM PRG_Semantic_Preservation_Governor
  VAR
    L_Now_MS : UDINT;
    L_Semantic_Valid : BOOL := TRUE;
    L_Error_Code : UDINT := 0;
    L_Error_Text : STRING(160) := '';
  END_VAR

            L_Now_MS := GVL_STATUS.G_System_Time_MS;
L_Semantic_Valid := TRUE;
L_Error_Code := 0;
L_Error_Text := '';

// Fail-safe defaults.
GVL_SEMANTIC_PRESERVATION_FABRIC.Semantic_Preservation_Valid := FALSE;
GVL_SEMANTIC_PRESERVATION_FABRIC.Semantic_Preservation_Granted := FALSE;
GVL_SEMANTIC_PRESERVATION_FABRIC.Semantic_Preservation_Quarantine_Active := TRUE;

GVL_SEMANTIC_PRESERVATION_FABRIC.Declared_System_Intent_Coherent := FALSE;
GVL_SEMANTIC_PRESERVATION_FABRIC.Adaptive_Policy_Bounded := FALSE;
GVL_SEMANTIC_PRESERVATION_FABRIC.Cross_Domain_Intent_Aligned := FALSE;
GVL_SEMANTIC_PRESERVATION_FABRIC.Optimization_Goals_Coherent := FALSE;
GVL_SEMANTIC_PRESERVATION_FABRIC.Behavioral_Evolution_Stable := FALSE;

// Runtime sustainability required.
IF NOT GVL_RUNTIME_SUSTAINABILITY_FABRIC.Runtime_Sustainability_Granted THEN
    L_Semantic_Valid := FALSE;
    L_Error_Code := 39000;
    L_Error_Text := 'Runtime sustainability authority not granted';
END_IF;

// Semantic drift detectors.
IF GVL_SEMANTIC_PRESERVATION_FABRIC.Adaptive_Policy_Drift_Detected THEN
    L_Semantic_Valid := FALSE;
    L_Error_Code := 39001;
    L_Error_Text := 'Adaptive policy drift detected';
END_IF;

IF GVL_SEMANTIC_PRESERVATION_FABRIC.Optimization_Semantic_Erosion_Detected THEN
    L_Semantic_Valid := FALSE;
    L_Error_Code := 39002;
    L_Error_Text := 'Optimization semantic erosion detected';
END_IF;

IF GVL_SEMANTIC_PRESERVATION_FABRIC.CrossDomain_Intent_Divergence_Detected THEN
    L_Semantic_Valid := FALSE;
    L_Error_Code := 39003;
    L_Error_Text := 'Cross-domain intent divergence detected';
END_IF;

IF GVL_SEMANTIC_PRESERVATION_FABRIC.LongTerm_Objective_Mutation_Detected THEN
    L_Semantic_Valid := FALSE;
    L_Error_Code := 39004;
    L_Error_Text := 'Long-term objective mutation detected';
END_IF;

IF GVL_SEMANTIC_PRESERVATION_FABRIC.Behavior_Learning_Instability_Detected THEN
    L_Semantic_Valid := FALSE;
    L_Error_Code := 39005;
    L_Error_Text := 'Behavior learning instability detected';
END_IF;

IF GVL_SEMANTIC_PRESERVATION_FABRIC.Silent_Governance_Reinterpretation_Detected THEN
    L_Semantic_Valid := FALSE;
    L_Error_Code := 39006;
    L_Error_Text := 'Silent governance reinterpretation detected';
END_IF;

// Immutable semantic intent validation.
IF L_Semantic_Valid
AND NOT GVL_SEMANTIC_PRESERVATION_FABRIC.Objective_Boundaries_Immutable THEN
    L_Semantic_Valid := FALSE;
    L_Error_Code := 39010;
    L_Error_Text := 'Objective boundaries immutability invalid';
END_IF;

IF L_Semantic_Valid
AND NOT GVL_SEMANTIC_PRESERVATION_FABRIC.Semantic_Governance_Coherent THEN
    L_Semantic_Valid := FALSE;
    L_Error_Code := 39011;
    L_Error_Text := 'Semantic governance coherence invalid';
END_IF;

IF L_Semantic_Valid
AND NOT GVL_SEMANTIC_PRESERVATION_FABRIC.Adaptive_Runtime_Intent_Stable THEN
    L_Semantic_Valid := FALSE;
    L_Error_Code := 39012;
    L_Error_Text := 'Adaptive runtime intent unstable';
END_IF;

IF L_Semantic_Valid
AND NOT GVL_SEMANTIC_PRESERVATION_FABRIC.LongTerm_Semantic_Evolution_Valid THEN
    L_Semantic_Valid := FALSE;
    L_Error_Code := 39013;
    L_Error_Text := 'Long-term semantic evolution invalid';
END_IF;

IF L_Semantic_Valid THEN
    GVL_SEMANTIC_PRESERVATION_FABRIC.Semantic_Preservation_Valid := TRUE;
    GVL_SEMANTIC_PRESERVATION_FABRIC.Semantic_Preservation_Granted := TRUE;
    GVL_SEMANTIC_PRESERVATION_FABRIC.Semantic_Preservation_Quarantine_Active := FALSE;

    GVL_SEMANTIC_PRESERVATION_FABRIC.Declared_System_Intent_Coherent := TRUE;
    GVL_SEMANTIC_PRESERVATION_FABRIC.Adaptive_Policy_Bounded := TRUE;
    GVL_SEMANTIC_PRESERVATION_FABRIC.Cross_Domain_Intent_Aligned := TRUE;
    GVL_SEMANTIC_PRESERVATION_FABRIC.Optimization_Goals_Coherent := TRUE;
    GVL_SEMANTIC_PRESERVATION_FABRIC.Behavioral_Evolution_Stable := TRUE;

    GVL_SEMANTIC_PRESERVATION_FABRIC.Semantic_Preservation_Epoch :=
        GVL_RUNTIME_SUSTAINABILITY_FABRIC.Runtime_Sustainability_Epoch;

    GVL_SEMANTIC_PRESERVATION_FABRIC.Semantic_Preservation_Epoch_Coherent := TRUE;

    GVL_SEMANTIC_PRESERVATION_FABRIC.Semantic_Preservation_Last_Update_MS :=
        L_Now_MS;

    GVL_SEMANTIC_PRESERVATION_FABRIC.Semantic_Preservation_Lease_Expired := FALSE;

    GVL_SEMANTIC_PRESERVATION_FABRIC.Semantic_Preservation_Last_Error_Code := 0;
    GVL_SEMANTIC_PRESERVATION_FABRIC.Semantic_Preservation_Last_Error_Text := '';
ELSE
    GVL_SEMANTIC_PRESERVATION_FABRIC.Semantic_Preservation_Valid := FALSE;
    GVL_SEMANTIC_PRESERVATION_FABRIC.Semantic_Preservation_Granted := FALSE;
    GVL_SEMANTIC_PRESERVATION_FABRIC.Semantic_Preservation_Quarantine_Active := TRUE;

    GVL_SEMANTIC_PRESERVATION_FABRIC.Semantic_Preservation_Lease_Expired := TRUE;

    GVL_SEMANTIC_PRESERVATION_FABRIC.Semantic_Preservation_Last_Error_Code :=
        L_Error_Code;

    GVL_SEMANTIC_PRESERVATION_FABRIC.Semantic_Preservation_Last_Error_Text :=
        L_Error_Text;

    GVL_SEMANTIC_PRESERVATION_FABRIC.Semantic_Preservation_Invalidation_Count :=
        GVL_SEMANTIC_PRESERVATION_FABRIC.Semantic_Preservation_Invalidation_Count + 1;
END_IF;
          
END_PROGRAM

PROGRAM PRG_Temporal_Domain

            // SEMANTIC DOMAIN WRAPPER
// PRESERVES ORIGINAL EXECUTION ORDER

PRG_Temporal_Stability_Governor();
PRG_Control_Temporal_Coherence_Governor();

PRG_Temporal_Causality_Closure_Governor();
PRG_Distributed_Epoch_Linearity_Governor();
PRG_Historical_Ordering_Integrity_Governor();
PRG_Causality_Reversal_Prevention_Governor();
          
END_PROGRAM

PROGRAM PRG_Safety
  VAR
    fbWaterLeakageManager : FB_Water_Leakage_Manager;
    fbGasSmokeManager : FB_Gas_Smoke_Manager;
    fbOwnership : FB_Ownership_Watchdog;
    L_i : INT;
  END_VAR

            GVL_INTENT_SAFETY.I_Source_Valid := TRUE;
GVL_INTENT_SAFETY.I_Last_Update_MS := GVL_TIME_SERVICE.G_Now_MS;
GVL_INTENT_SAFETY.I_Fire_Alarm_Active := FALSE;
GVL_INTENT_SAFETY.I_Gas_Alarm_Active := FALSE;
GVL_INTENT_SAFETY.I_Leak_Alarm_Active := FALSE;
GVL_INTENT_SAFETY.I_CO_Warning_Active := FALSE;
GVL_INTENT_SAFETY.I_System_Safe_Stop_Required := FALSE;
GVL_INTENT_SAFETY.I_Freeze_Protection_Required := FALSE;
GVL_INTENT_SAFETY.I_Evacuation_Mode_Active := FALSE;
GVL_INTENT_SAFETY.I_Gas_Close_Required := FALSE;
GVL_INTENT_SAFETY.I_Boiler_Stop_Required := FALSE;
GVL_INTENT_SAFETY.I_Vent_Stop_Required := FALSE;
GVL_INTENT_SAFETY.I_Vent_Force_PV3_Boost := FALSE;
GVL_INTENT_SAFETY.I_Vent_Force_Supply_100 := FALSE;
GVL_INTENT_SAFETY.I_Vent_Force_Supply_80 := FALSE;
GVL_INTENT_SAFETY.I_Vent_Force_Exhaust_100 := FALSE;
GVL_INTENT_SAFETY.I_Water_Main_Close_Required := FALSE;
GVL_INTENT_SAFETY.I_Water_Selective_Recovery_Allowed := FALSE;
GVL_INTENT_SAFETY.I_Water_Recovery_Target_Zone := 0;
GVL_INTENT_SAFETY.I_Lock_1_Force_Open := FALSE;
GVL_INTENT_SAFETY.I_Lock_1_Force_Close_Block := FALSE;
GVL_INTENT_SAFETY.I_Lock_2_Force_Open := FALSE;
GVL_INTENT_SAFETY.I_Lock_2_Force_Close_Block := FALSE;

fbWaterLeakageManager(
    VI_System_Time_MS := GVL_TIME_SERVICE.G_Now_MS,
    VI_IsActivePLC := GVL_STATUS.G_Is_Active_PLC,
    VI_Sensors := GVL_STATE.G_Water_Sensors,
    VI_Config := GVL_CONFIG.G_HMI_Flood_Config,
    VO_Status_Msg => GVL_STATUS.G_Flood_Status_Msg,
    VO_Leak_Detected => GVL_HEALTH_BRIDGE.G_Leak_Detected,
    VO_Leak_Warning_Level => GVL_HEALTH_BRIDGE.G_Leak_Warning_Level
);
GVL_INTENT_SAFETY.I_Leak_Alarm_Active := GVL_HEALTH_BRIDGE.G_Leak_Detected;

fbGasSmokeManager(
    VI_System_Time_MS := GVL_TIME_SERVICE.G_Now_MS,
    VI_IsActivePLC := GVL_STATUS.G_Is_Active_PLC,
    VI_Methane_LEL := GVL_Safety_Selector.G_Methane_Effective_Array,
    VI_CO_PPM := GVL_Safety_Selector.G_CO_Effective_Array,
    VI_Smoke_Sensors := GVL_Safety_Selector.G_Smoke_Effective_Array,
    VI_Mute_Request := GVL_CONFIG.G_HMI_Mute_Alarm,
    VO_Smoke_Detected => GVL_HEALTH_BRIDGE.G_Smoke_Detected,
    VO_Gas_Detected => GVL_HEALTH_BRIDGE.G_Gas_Detected,
    VO_CO_Warning_Level => GVL_HEALTH_BRIDGE.G_CO_Warning_Level,
    VO_CO_Alarm_Level => GVL_HEALTH_BRIDGE.G_CO_Alarm_Level,
    VO_Status_Msg => GVL_STATUS.G_Gas_Status_Msg
);
GVL_INTENT_SAFETY.I_Fire_Alarm_Active := GVL_HEALTH_BRIDGE.G_Smoke_Detected;
GVL_INTENT_SAFETY.I_Gas_Alarm_Active := GVL_HEALTH_BRIDGE.G_Gas_Detected OR GVL_HEALTH_BRIDGE.G_CO_Alarm_Level;
GVL_INTENT_SAFETY.I_CO_Warning_Active := GVL_HEALTH_BRIDGE.G_CO_Warning_Level;

// Ownership watchdog must observe authoritative safety truth, not stale
// projected GVL_STATE.G_Safety_*_Alarm compatibility fields.
fbOwnership(
    VI_Gas_Level := GVL_Safety_Selector.G_Methane_Effective_Array[GVL_CONSTANTS.C_PRIMARY_EFFECTIVE_GAS_INDEX],
    VI_Gas_Alarm := GVL_HEALTH_BRIDGE.G_Gas_Detected OR GVL_HEALTH_BRIDGE.G_CO_Alarm_Level,
    VI_Leak_Alarm := GVL_HEALTH_BRIDGE.G_Leak_Detected,
    VI_Smoke_Alarm := GVL_HEALTH_BRIDGE.G_Smoke_Detected
);

IF fbOwnership.VO_Ownership_Violation THEN
    GVL_DEBUG_VIEW.D_Ownership_Violation := TRUE;
END_IF;

IF GVL_STATE.G_Safety_Smoke_Latched THEN
    GVL_INTENT_SAFETY.I_System_Safe_Stop_Required := TRUE;
    GVL_INTENT_SAFETY.I_Evacuation_Mode_Active := TRUE;
    GVL_INTENT_SAFETY.I_Boiler_Stop_Required := TRUE;
    GVL_INTENT_SAFETY.I_Vent_Stop_Required := TRUE;
    GVL_INTENT_SAFETY.I_Lock_1_Force_Open := TRUE;
    GVL_INTENT_SAFETY.I_Lock_1_Force_Close_Block := TRUE;
    GVL_INTENT_SAFETY.I_Lock_2_Force_Open := TRUE;
    GVL_INTENT_SAFETY.I_Lock_2_Force_Close_Block := TRUE;
END_IF;

IF GVL_STATE.G_Safety_Gas_Latched THEN
    GVL_INTENT_SAFETY.I_System_Safe_Stop_Required := TRUE;
    GVL_INTENT_SAFETY.I_Gas_Close_Required := TRUE;
    GVL_INTENT_SAFETY.I_Boiler_Stop_Required := TRUE;
    GVL_INTENT_SAFETY.I_Vent_Force_PV3_Boost := TRUE;
    GVL_INTENT_SAFETY.I_Vent_Force_Supply_100 := TRUE;
END_IF;

IF GVL_HEALTH_BRIDGE.G_CO_Warning_Level OR GVL_HEALTH_BRIDGE.G_CO_Alarm_Level THEN
    GVL_INTENT_SAFETY.I_Vent_Force_Supply_80 := TRUE;
END_IF;

IF GVL_STATE.G_Safety_Leak_Latched THEN
    GVL_INTENT_SAFETY.I_Water_Main_Close_Required := TRUE;
END_IF;

IF GVL_STATE.G_Freeze_Hardware_Degraded THEN
    GVL_INTENT_SAFETY.I_Freeze_Protection_Required := TRUE;
END_IF;

// >>> BULK_SYNC_ANCHOR: PRG_Safety <<<
          
END_PROGRAM

PROGRAM PRG_Telemetry_Causality_Governor
  VAR
    L_Now_MS : UDINT;
    L_Causality_Valid : BOOL := TRUE;
    L_Error_Code : UDINT := 0;
    L_Error_Text : STRING(160) := '';
    L_Ack_Age_MS : UDINT;
    L_Convergence_Age_MS : UDINT;
    L_Stable_Dwell_MS : UDINT;
    L_Consensus_Age_MS : UDINT;
  END_VAR

            L_Now_MS := GVL_STATUS.G_System_Time_MS;
L_Causality_Valid := TRUE;
L_Error_Code := 0;
L_Error_Text := '';

GVL_TELEMETRY.Telemetry_Runtime_Valid := FALSE;
GVL_TELEMETRY.Telemetry_Freshness_Valid := FALSE;
GVL_TELEMETRY.Command_Telemetry_Causality_Valid := FALSE;
GVL_TELEMETRY.Actuator_Feedback_Valid := FALSE;
GVL_TELEMETRY.Actuator_Feedback_Fresh := FALSE;
GVL_TELEMETRY.Physical_Effect_Confirmed := FALSE;
GVL_TELEMETRY.Physical_Effect_Finalized := FALSE;
GVL_TELEMETRY.Physical_Target_Converged := FALSE;
GVL_TELEMETRY.Physical_Stable_Window_OK := FALSE;
GVL_TELEMETRY.Command_Telemetry_Divergence_Detected := TRUE;

GVL_TELEMETRY.Command_Epoch := ULINT_TO_UDINT(GVL_OUTPUT_EPOCH.Output_Publication_Epoch);

IF NOT GVL_OUTPUT_EPOCH.Output_Publication_Valid THEN
    L_Causality_Valid := FALSE;
    L_Error_Code := 21000;
    L_Error_Text := 'Telemetry causality output publication invalid';
END_IF;

IF L_Causality_Valid AND NOT GVL_OUTPUT_EPOCH.Output_Runtime_Epoch_Valid THEN
    L_Causality_Valid := FALSE;
    L_Error_Code := 21001;
    L_Error_Text := 'Telemetry causality runtime epoch invalid';
END_IF;

IF L_Causality_Valid AND GVL_OUTPUT_EPOCH.Output_Lease_Expired THEN
    L_Causality_Valid := FALSE;
    L_Error_Code := 21002;
    L_Error_Text := 'Telemetry causality output lease expired';
END_IF;

IF L_Causality_Valid AND GVL_OUTPUT_EPOCH.Output_Forced_Safe_Decay THEN
    L_Causality_Valid := FALSE;
    L_Error_Code := 21003;
    L_Error_Text := 'Telemetry causality output forced safe decay';
END_IF;

IF L_Causality_Valid AND (GVL_TELEMETRY.Telemetry_Epoch <> GVL_TELEMETRY.Command_Epoch) THEN
    L_Causality_Valid := FALSE;
    L_Error_Code := 21010;
    L_Error_Text := 'Telemetry epoch does not match command epoch';
END_IF;

IF L_Causality_Valid AND (GVL_TELEMETRY.Telemetry_Epoch < GVL_TELEMETRY.Last_Acknowledged_Command_Epoch) THEN
    GVL_TELEMETRY.Telemetry_Replay_Suspected := TRUE;

    L_Causality_Valid := FALSE;
    L_Error_Code := 21011;
    L_Error_Text := 'Telemetry epoch replay suspected';
END_IF;

L_Ack_Age_MS := L_Now_MS - GVL_TELEMETRY.Last_Physical_Ack_Time_MS;

IF L_Causality_Valid AND (L_Ack_Age_MS > 5000) THEN
    L_Causality_Valid := FALSE;
    L_Error_Code := 21020;
    L_Error_Text := 'Physical acknowledgement stale';
END_IF;

L_Convergence_Age_MS := L_Now_MS - GVL_TELEMETRY.Last_Physical_Convergence_MS;

IF L_Causality_Valid AND (L_Convergence_Age_MS > 10000) THEN
    L_Causality_Valid := FALSE;
    L_Error_Code := 21021;
    L_Error_Text := 'Physical convergence stale';
END_IF;

L_Stable_Dwell_MS :=
    L_Now_MS - GVL_TELEMETRY.Last_Physical_Convergence_MS;

IF L_Causality_Valid AND (L_Stable_Dwell_MS < 3000) THEN
    L_Causality_Valid := FALSE;
    L_Error_Code := 21030;
    L_Error_Text := 'Physical stabilization dwell window incomplete';
END_IF;

IF L_Causality_Valid
AND GVL_TELEMETRY.Physical_Oscillation_Detected THEN
    L_Causality_Valid := FALSE;
    L_Error_Code := 21031;
    L_Error_Text := 'Physical oscillation detected';
END_IF;

IF L_Causality_Valid
AND GVL_TELEMETRY.Physical_Transition_Active THEN
    L_Causality_Valid := FALSE;
    L_Error_Code := 21032;
    L_Error_Text := 'Physical transition still active';
END_IF;

IF L_Causality_Valid
AND GVL_TELEMETRY.Physical_Convergence_Replay_Suspected THEN
    L_Causality_Valid := FALSE;
    L_Error_Code := 21033;
    L_Error_Text := 'Physical convergence replay suspected';
END_IF;

L_Consensus_Age_MS :=
    L_Now_MS - GVL_SENSOR_CONSENSUS.Last_Consensus_Update_MS;

IF L_Causality_Valid
AND (L_Consensus_Age_MS > 5000) THEN
    L_Causality_Valid := FALSE;
    L_Error_Code := 21040;
    L_Error_Text := 'Sensor consensus stale';
END_IF;

IF L_Causality_Valid
AND NOT GVL_SENSOR_CONSENSUS.Sensor_Consensus_Valid THEN
    L_Causality_Valid := FALSE;
    L_Error_Code := 21041;
    L_Error_Text := 'Sensor consensus invalid';
END_IF;

IF L_Causality_Valid
AND NOT GVL_SENSOR_CONSENSUS.Physics_Invariants_Satisfied THEN
    L_Causality_Valid := FALSE;
    L_Error_Code := 21042;
    L_Error_Text := 'Physics invariants violated';
END_IF;

IF L_Causality_Valid
AND NOT GVL_SENSOR_CONSENSUS.Cross_Sensor_Correlation_Valid THEN
    L_Causality_Valid := FALSE;
    L_Error_Code := 21043;
    L_Error_Text := 'Cross sensor correlation invalid';
END_IF;

IF L_Causality_Valid
AND NOT GVL_SENSOR_CONSENSUS.Telemetry_Plausibility_Valid THEN
    L_Causality_Valid := FALSE;
    L_Error_Code := 21044;
    L_Error_Text := 'Telemetry plausibility invalid';
END_IF;

IF L_Causality_Valid
AND (GVL_SENSOR_CONSENSUS.Sensor_Drift_Detected
     OR GVL_SENSOR_CONSENSUS.Sensor_Partition_Detected
     OR GVL_SENSOR_CONSENSUS.Sensor_Hallucination_Suspected
     OR GVL_SENSOR_CONSENSUS.Cross_Sensor_Divergence_Detected
     OR GVL_SENSOR_CONSENSUS.Sensor_Oscillation_Detected
     OR GVL_SENSOR_CONSENSUS.Sensor_Stuck_State_Detected
     OR GVL_SENSOR_CONSENSUS.Sensor_Replay_Suspected) THEN

    L_Causality_Valid := FALSE;
    L_Error_Code := 21045;
    L_Error_Text := 'Sensor consensus divergence detected';
END_IF;

IF L_Causality_Valid THEN
    GVL_TELEMETRY.Telemetry_Runtime_Valid := TRUE;
    GVL_TELEMETRY.Telemetry_Freshness_Valid := TRUE;
    GVL_TELEMETRY.Telemetry_Lease_Expired := FALSE;
    GVL_TELEMETRY.Telemetry_Quarantine_Active := FALSE;

    GVL_TELEMETRY.Command_Telemetry_Causality_Valid := TRUE;
    GVL_TELEMETRY.Command_Telemetry_Divergence_Detected := FALSE;

    GVL_TELEMETRY.Actuator_Feedback_Valid := TRUE;
    GVL_TELEMETRY.Actuator_Feedback_Fresh := TRUE;
    GVL_TELEMETRY.Physical_Effect_Confirmed := TRUE;

    GVL_TELEMETRY.Physical_Target_Converged := TRUE;
    GVL_TELEMETRY.Physical_Stable_Window_OK := TRUE;
    GVL_TELEMETRY.Physical_Effect_Finalized := TRUE;

    GVL_TELEMETRY.Last_Acknowledged_Command_Epoch := GVL_TELEMETRY.Command_Epoch;

    GVL_TELEMETRY.Telemetry_Last_Error_Code := 0;
    GVL_TELEMETRY.Telemetry_Last_Error_Text := '';
ELSE
    GVL_TELEMETRY.Telemetry_Runtime_Valid := FALSE;
    GVL_TELEMETRY.Telemetry_Freshness_Valid := FALSE;
    GVL_TELEMETRY.Telemetry_Lease_Expired := TRUE;
    GVL_TELEMETRY.Telemetry_Quarantine_Active := TRUE;

    GVL_TELEMETRY.Command_Telemetry_Causality_Valid := FALSE;
    GVL_TELEMETRY.Command_Telemetry_Divergence_Detected := TRUE;

    GVL_TELEMETRY.Telemetry_Last_Error_Code := L_Error_Code;
    GVL_TELEMETRY.Telemetry_Last_Error_Text := L_Error_Text;
    GVL_TELEMETRY.Telemetry_Invalidation_Count :=
        GVL_TELEMETRY.Telemetry_Invalidation_Count + 1;
END_IF;
          
END_PROGRAM

PROGRAM PRG_Historical_Truth_Governor
  VAR
    L_Now_MS : UDINT;
    L_History_Valid : BOOL := TRUE;
    L_Error_Code : UDINT := 0;
    L_Error_Text : STRING(160) := '';
  END_VAR

            L_Now_MS := GVL_STATUS.G_System_Time_MS;
L_History_Valid := TRUE;
L_Error_Code := 0;
L_Error_Text := '';

// Fail-safe defaults.
GVL_HISTORICAL_TRUTH.Historical_Truth_Valid := FALSE;
GVL_HISTORICAL_TRUTH.Historical_Truth_Granted := FALSE;
GVL_HISTORICAL_TRUTH.Historical_Truth_Quarantine_Active := TRUE;

GVL_HISTORICAL_TRUTH.Trend_History_Causally_Immutable := FALSE;
GVL_HISTORICAL_TRUTH.Alarm_Chronology_Immutable := FALSE;
GVL_HISTORICAL_TRUTH.Blackbox_Snapshot_Immutable := FALSE;
GVL_HISTORICAL_TRUTH.Diagnostics_History_Coherent := FALSE;
GVL_HISTORICAL_TRUTH.Failover_Chronology_Coherent := FALSE;

// Observability truth authority required.
IF NOT GVL_OBSERVABILITY_TRUTH.Observability_Truth_Granted THEN
    L_History_Valid := FALSE;
    L_Error_Code := 33000;
    L_Error_Text := 'Observability truth authority not granted';
END_IF;

// Historical corruption detectors.
IF GVL_HISTORICAL_TRUTH.History_Epoch_Skew_Detected THEN
    L_History_Valid := FALSE;
    L_Error_Code := 33001;
    L_Error_Text := 'Historical epoch skew detected';
END_IF;

IF GVL_HISTORICAL_TRUTH.Failover_Chronology_Corruption_Detected THEN
    L_History_Valid := FALSE;
    L_Error_Code := 33002;
    L_Error_Text := 'Failover chronology corruption detected';
END_IF;

IF GVL_HISTORICAL_TRUTH.Trend_Replay_Race_Detected THEN
    L_History_Valid := FALSE;
    L_Error_Code := 33003;
    L_Error_Text := 'Trend replay race detected';
END_IF;

IF GVL_HISTORICAL_TRUTH.Blackbox_Causality_Drift_Detected THEN
    L_History_Valid := FALSE;
    L_Error_Code := 33004;
    L_Error_Text := 'Blackbox causality drift detected';
END_IF;

IF GVL_HISTORICAL_TRUTH.Alarm_Order_Reconstruction_Error THEN
    L_History_Valid := FALSE;
    L_Error_Code := 33005;
    L_Error_Text := 'Alarm order reconstruction error detected';
END_IF;

IF GVL_HISTORICAL_TRUTH.Mixed_Authority_Persistence_Detected THEN
    L_History_Valid := FALSE;
    L_Error_Code := 33006;
    L_Error_Text := 'Mixed-authority persistence detected';
END_IF;

// Historical persistence integrity validation.
IF L_History_Valid
AND NOT GVL_HISTORICAL_TRUTH.Persisted_Epochs_Coherent THEN
    L_History_Valid := FALSE;
    L_Error_Code := 33010;
    L_Error_Text := 'Persisted epoch coherence invalid';
END_IF;

IF L_History_Valid
AND NOT GVL_HISTORICAL_TRUTH.Recovery_Replay_Coherent THEN
    L_History_Valid := FALSE;
    L_Error_Code := 33011;
    L_Error_Text := 'Recovery replay coherence invalid';
END_IF;

IF L_History_Valid
AND NOT GVL_HISTORICAL_TRUTH.Historical_Snapshot_Coherent THEN
    L_History_Valid := FALSE;
    L_Error_Code := 33012;
    L_Error_Text := 'Historical snapshot coherence invalid';
END_IF;

IF L_History_Valid
AND NOT GVL_HISTORICAL_TRUTH.Mixed_Authority_Persistence_Absent THEN
    L_History_Valid := FALSE;
    L_Error_Code := 33013;
    L_Error_Text := 'Mixed-authority persistence absence invalid';
END_IF;

IF L_History_Valid THEN
    GVL_HISTORICAL_TRUTH.Historical_Truth_Valid := TRUE;
    GVL_HISTORICAL_TRUTH.Historical_Truth_Granted := TRUE;
    GVL_HISTORICAL_TRUTH.Historical_Truth_Quarantine_Active := FALSE;

    GVL_HISTORICAL_TRUTH.Trend_History_Causally_Immutable := TRUE;
    GVL_HISTORICAL_TRUTH.Alarm_Chronology_Immutable := TRUE;
    GVL_HISTORICAL_TRUTH.Blackbox_Snapshot_Immutable := TRUE;
    GVL_HISTORICAL_TRUTH.Diagnostics_History_Coherent := TRUE;
    GVL_HISTORICAL_TRUTH.Failover_Chronology_Coherent := TRUE;

    GVL_HISTORICAL_TRUTH.Historical_Truth_Epoch :=
        GVL_OBSERVABILITY_TRUTH.Observability_Truth_Epoch;

    GVL_HISTORICAL_TRUTH.Historical_Truth_Epoch_Coherent := TRUE;

    GVL_HISTORICAL_TRUTH.Historical_Last_Update_MS := L_Now_MS;
    GVL_HISTORICAL_TRUTH.Historical_Lease_Expired := FALSE;

    GVL_HISTORICAL_TRUTH.Historical_Last_Error_Code := 0;
    GVL_HISTORICAL_TRUTH.Historical_Last_Error_Text := '';
ELSE
    GVL_HISTORICAL_TRUTH.Historical_Truth_Valid := FALSE;
    GVL_HISTORICAL_TRUTH.Historical_Truth_Granted := FALSE;
    GVL_HISTORICAL_TRUTH.Historical_Truth_Quarantine_Active := TRUE;

    GVL_HISTORICAL_TRUTH.Historical_Lease_Expired := TRUE;

    GVL_HISTORICAL_TRUTH.Historical_Last_Error_Code :=
        L_Error_Code;

    GVL_HISTORICAL_TRUTH.Historical_Last_Error_Text :=
        L_Error_Text;

    GVL_HISTORICAL_TRUTH.Historical_Invalidation_Count :=
        GVL_HISTORICAL_TRUTH.Historical_Invalidation_Count + 1;
END_IF;
          
END_PROGRAM

PROGRAM PRG_Unsafe_Transition_Forensics_Governor

            IF GVL_PHYSICAL_SAFETY_PROJECTION_FABRIC.Physical_Safety_Projection_Granted
AND NOT GVL_UNSAFE_TRANSITION_FORENSICS_FABRIC.Unsafe_Transition_Hidden
AND NOT GVL_UNSAFE_TRANSITION_FORENSICS_FABRIC.Forensic_Lineage_Break_Detected
AND NOT GVL_UNSAFE_TRANSITION_FORENSICS_FABRIC.Historical_Safety_Gap_Detected THEN

    GVL_UNSAFE_TRANSITION_FORENSICS_FABRIC.Unsafe_Transition_Forensics_Valid := TRUE;
    GVL_UNSAFE_TRANSITION_FORENSICS_FABRIC.Unsafe_Transition_Forensics_Granted := TRUE;
    GVL_UNSAFE_TRANSITION_FORENSICS_FABRIC.Unsafe_Transition_Lineage_Preserved := TRUE;
    GVL_UNSAFE_TRANSITION_FORENSICS_FABRIC.Forensic_Causality_Continuity_Valid := TRUE;
    GVL_UNSAFE_TRANSITION_FORENSICS_FABRIC.Distributed_Unsafe_Event_Consensus := TRUE;
END_IF;
          
END_PROGRAM

PROGRAM PRG_Input_Quality_Read
  VAR
    L_i : INT;
    fbRoomTempQuality : ARRAY[1..GVL_CONSTANTS.C_MAX_ZONES] OF FB_Input_Quality_Observer;
    fbFloorTempQuality : ARRAY[1..GVL_CONSTANTS.C_MAX_HEATING_CIRCUITS] OF FB_Input_Quality_Observer;
  END_VAR

            FOR L_i := 1 TO GVL_CONSTANTS.C_MAX_ZONES DO
    fbRoomTempQuality[L_i](
        VI_Enable := GVL_INPUT_VALIDATION_CONFIG.G_Enable_Temporal_Anomaly_Detection,
        VI_Value := GVL_STATE.G_Room_Temps[L_i],
        VI_System_Time_MS := GVL_STATUS.G_System_Time_MS,
        VI_Spike_Threshold := GVL_INPUT_VALIDATION_CONFIG.G_Room_Temp_Spike_Threshold,
        VI_Stuck_Timeout_MS := GVL_INPUT_VALIDATION_CONFIG.G_Sensor_Stuck_Timeout_MS,
        VO_Quality => GVL_INPUT_QUALITY.G_Room_Temp_Quality[L_i]
    );
END_FOR;

FOR L_i := 1 TO GVL_CONSTANTS.C_MAX_HEATING_CIRCUITS DO
    fbFloorTempQuality[L_i](
        VI_Enable := GVL_INPUT_VALIDATION_CONFIG.G_Enable_Temporal_Anomaly_Detection,
        VI_Value := GVL_STATE.G_Floor_Temps[L_i],
        VI_System_Time_MS := GVL_STATUS.G_System_Time_MS,
        VI_Spike_Threshold := GVL_INPUT_VALIDATION_CONFIG.G_Room_Temp_Spike_Threshold,
        VI_Stuck_Timeout_MS := GVL_INPUT_VALIDATION_CONFIG.G_Sensor_Stuck_Timeout_MS,
        VO_Quality => GVL_INPUT_QUALITY.G_Floor_Temp_Quality[L_i]
    );
END_FOR;
          
END_PROGRAM

PROGRAM PRG_Controlled_Capability_Shedding_Governor

            // CONTROLLED CAPABILITY SHEDDING
// DETERMINISTIC / TIER-AWARE / NON-INVASIVE

IF GVL_RUNTIME_BUDGET_ENFORCEMENT.Runtime_Budget_Pressure_Observed THEN
    GVL_FABRIC_LIFECYCLE_REGISTRY.Controlled_Capability_Shedding_Allowed := TRUE;
    GVL_FABRIC_LIFECYCLE_REGISTRY.Runtime_Adaptive_Mode := REDUCED_ANALYTICS_MODE;
END_IF;

IF GVL_SURVIVABILITY_INTELLIGENCE_FABRIC.Chronic_Degradation_Risk_Increasing THEN
    GVL_FABRIC_LIFECYCLE_REGISTRY.Runtime_Adaptive_Mode := SURVIVABILITY_MODE;
    GVL_FABRIC_LIFECYCLE_REGISTRY.NonEssential_Analytics_Shedding_Recommended := TRUE;
    GVL_FABRIC_LIFECYCLE_REGISTRY.Diagnostics_Degradation_Recommended := TRUE;
END_IF;

IF GVL_RUNTIME_BUDGET_ENFORCEMENT.Verification_Induced_Runtime_Risk THEN
    GVL_FABRIC_LIFECYCLE_REGISTRY.Extended_Observability_Shedding_Recommended := TRUE;
    GVL_FABRIC_LIFECYCLE_REGISTRY.Simulation_Suspension_Recommended := TRUE;
END_IF;

IF GVL_RUNTIME_BUDGET_ENFORCEMENT.Runtime_Stability_Budget_At_Risk THEN
    GVL_FABRIC_LIFECYCLE_REGISTRY.Analytics_Fabric_State := FABRIC_DEGRADED;
    GVL_FABRIC_LIFECYCLE_REGISTRY.Observability_Fabric_State := FABRIC_PASSIVE;
END_IF;

// Critical fabrics remain protected.
GVL_FABRIC_LIFECYCLE_REGISTRY.Safety_Fabric_State := FABRIC_ACTIVE;
GVL_FABRIC_LIFECYCLE_REGISTRY.Authority_Fabric_State := FABRIC_ACTIVE;
GVL_FABRIC_LIFECYCLE_REGISTRY.Physical_Reality_Fabric_State := FABRIC_ACTIVE;

IF NOT GVL_RUNTIME_BUDGET_ENFORCEMENT.Runtime_Budget_Pressure_Observed THEN
    GVL_FABRIC_LIFECYCLE_REGISTRY.Gradual_Reactivation_Allowed := TRUE;
END_IF;
          
END_PROGRAM

PROGRAM PRG_Runtime_Core_Domain

            // CANONICAL EXECUTION DOMAIN
// PRESERVES EXECUTION ORDER

PRG_Time_Service();
PRG_System_Init();
PRG_Runtime_Barrier();
PRG_Runtime_Snapshot_Governor();
PRG_Runtime_Assumption_Integrity_Governor();
          
END_PROGRAM

PROGRAM PRG_Runtime_Resource_Authority_Governor
  VAR
    L_Now_MS : UDINT;
    L_Runtime_Valid : BOOL := TRUE;
    L_Error_Code : UDINT := 0;
    L_Error_Text : STRING(160) := '';
  END_VAR

            L_Now_MS := GVL_STATUS.G_System_Time_MS;
L_Runtime_Valid := TRUE;
L_Error_Code := 0;
L_Error_Text := '';

// Fail-safe defaults.
GVL_RUNTIME_RESOURCE_AUTHORITY.Runtime_Resource_Authority_Valid := FALSE;
GVL_RUNTIME_RESOURCE_AUTHORITY.Runtime_Resource_Authority_Granted := FALSE;
GVL_RUNTIME_RESOURCE_AUTHORITY.Runtime_Resource_Quarantine_Active := TRUE;

GVL_RUNTIME_RESOURCE_AUTHORITY.Deterministic_Cycle_Time_Valid := FALSE;
GVL_RUNTIME_RESOURCE_AUTHORITY.Task_Jitter_Within_Bounds := FALSE;
GVL_RUNTIME_RESOURCE_AUTHORITY.Watchdog_Margin_Stable := FALSE;
GVL_RUNTIME_RESOURCE_AUTHORITY.Runtime_Latency_Stable := FALSE;
GVL_RUNTIME_RESOURCE_AUTHORITY.Queue_Backlog_Stable := FALSE;

// Environmental authority required.
IF NOT GVL_ENVIRONMENTAL_AUTHORITY.Environmental_Authority_Granted THEN
    L_Runtime_Valid := FALSE;
    L_Error_Code := 30000;
    L_Error_Text := 'Environmental authority not granted';
END_IF;

// Resource exhaustion detectors.
IF GVL_RUNTIME_RESOURCE_AUTHORITY.Hidden_Jitter_Amplification_Detected THEN
    L_Runtime_Valid := FALSE;
    L_Error_Code := 30001;
    L_Error_Text := 'Hidden jitter amplification detected';
END_IF;

IF GVL_RUNTIME_RESOURCE_AUTHORITY.Queue_Induced_Authority_Lag_Detected THEN
    L_Runtime_Valid := FALSE;
    L_Error_Code := 30002;
    L_Error_Text := 'Queue-induced authority lag detected';
END_IF;

IF GVL_RUNTIME_RESOURCE_AUTHORITY.Watchdog_Near_Death_Oscillation_Detected THEN
    L_Runtime_Valid := FALSE;
    L_Error_Code := 30003;
    L_Error_Text := 'Watchdog near-death oscillation detected';
END_IF;

IF GVL_RUNTIME_RESOURCE_AUTHORITY.Runtime_Starvation_Race_Detected THEN
    L_Runtime_Valid := FALSE;
    L_Error_Code := 30004;
    L_Error_Text := 'Runtime starvation race detected';
END_IF;

IF GVL_RUNTIME_RESOURCE_AUTHORITY.Cycle_Collapse_SplitBrain_Detected THEN
    L_Runtime_Valid := FALSE;
    L_Error_Code := 30005;
    L_Error_Text := 'Cycle collapse split-brain detected';
END_IF;

IF GVL_RUNTIME_RESOURCE_AUTHORITY.Heap_Fragmentation_Critical THEN
    L_Runtime_Valid := FALSE;
    L_Error_Code := 30006;
    L_Error_Text := 'Critical heap fragmentation detected';
END_IF;

IF GVL_RUNTIME_RESOURCE_AUTHORITY.Fieldbus_Backlog_Saturation_Detected THEN
    L_Runtime_Valid := FALSE;
    L_Error_Code := 30007;
    L_Error_Text := 'Fieldbus backlog saturation detected';
END_IF;

// Deterministic execution envelope validation.
IF L_Runtime_Valid
AND (GVL_RUNTIME_RESOURCE_AUTHORITY.Current_Task_Jitter_US >
     GVL_RUNTIME_RESOURCE_AUTHORITY.Max_Allowed_Task_Jitter_US) THEN

    L_Runtime_Valid := FALSE;
    L_Error_Code := 30010;
    L_Error_Text := 'Task jitter exceeds deterministic envelope';
END_IF;

IF L_Runtime_Valid
AND (GVL_RUNTIME_RESOURCE_AUTHORITY.Current_Runtime_Latency_US >
     GVL_RUNTIME_RESOURCE_AUTHORITY.Max_Allowed_Runtime_Latency_US) THEN

    L_Runtime_Valid := FALSE;
    L_Error_Code := 30011;
    L_Error_Text := 'Runtime latency exceeds deterministic envelope';
END_IF;

IF L_Runtime_Valid
AND (GVL_RUNTIME_RESOURCE_AUTHORITY.Current_Fieldbus_Queue_Depth >
     GVL_RUNTIME_RESOURCE_AUTHORITY.Max_Allowed_Fieldbus_Queue_Depth) THEN

    L_Runtime_Valid := FALSE;
    L_Error_Code := 30012;
    L_Error_Text := 'Fieldbus queue depth exceeds deterministic envelope';
END_IF;

IF L_Runtime_Valid
AND (GVL_RUNTIME_RESOURCE_AUTHORITY.Current_Watchdog_Margin_MS <
     GVL_RUNTIME_RESOURCE_AUTHORITY.Minimum_Watchdog_Margin_MS) THEN

    L_Runtime_Valid := FALSE;
    L_Error_Code := 30013;
    L_Error_Text := 'Watchdog margin below deterministic envelope';
END_IF;

IF L_Runtime_Valid THEN
    GVL_RUNTIME_RESOURCE_AUTHORITY.Runtime_Resource_Authority_Valid := TRUE;
    GVL_RUNTIME_RESOURCE_AUTHORITY.Runtime_Resource_Authority_Granted := TRUE;
    GVL_RUNTIME_RESOURCE_AUTHORITY.Runtime_Resource_Quarantine_Active := FALSE;

    GVL_RUNTIME_RESOURCE_AUTHORITY.Deterministic_Cycle_Time_Valid := TRUE;
    GVL_RUNTIME_RESOURCE_AUTHORITY.Task_Jitter_Within_Bounds := TRUE;
    GVL_RUNTIME_RESOURCE_AUTHORITY.Watchdog_Margin_Stable := TRUE;
    GVL_RUNTIME_RESOURCE_AUTHORITY.Runtime_Latency_Stable := TRUE;
    GVL_RUNTIME_RESOURCE_AUTHORITY.Queue_Backlog_Stable := TRUE;

    GVL_RUNTIME_RESOURCE_AUTHORITY.Runtime_Resource_Authority_Epoch :=
        GVL_ENVIRONMENTAL_AUTHORITY.Environmental_Authority_Epoch;

    GVL_RUNTIME_RESOURCE_AUTHORITY.Runtime_Resource_Authority_Epoch_Coherent := TRUE;

    GVL_RUNTIME_RESOURCE_AUTHORITY.Runtime_Resource_Last_Update_MS :=
        L_Now_MS;

    GVL_RUNTIME_RESOURCE_AUTHORITY.Runtime_Resource_Lease_Expired := FALSE;

    GVL_RUNTIME_RESOURCE_AUTHORITY.Runtime_Resource_Last_Error_Code := 0;
    GVL_RUNTIME_RESOURCE_AUTHORITY.Runtime_Resource_Last_Error_Text := '';
ELSE
    GVL_RUNTIME_RESOURCE_AUTHORITY.Runtime_Resource_Authority_Valid := FALSE;
    GVL_RUNTIME_RESOURCE_AUTHORITY.Runtime_Resource_Authority_Granted := FALSE;
    GVL_RUNTIME_RESOURCE_AUTHORITY.Runtime_Resource_Quarantine_Active := TRUE;

    GVL_RUNTIME_RESOURCE_AUTHORITY.Runtime_Resource_Lease_Expired := TRUE;

    GVL_RUNTIME_RESOURCE_AUTHORITY.Runtime_Resource_Last_Error_Code :=
        L_Error_Code;

    GVL_RUNTIME_RESOURCE_AUTHORITY.Runtime_Resource_Last_Error_Text :=
        L_Error_Text;

    GVL_RUNTIME_RESOURCE_AUTHORITY.Runtime_Resource_Invalidation_Count :=
        GVL_RUNTIME_RESOURCE_AUTHORITY.Runtime_Resource_Invalidation_Count + 1;
END_IF;
          
END_PROGRAM

PROGRAM PRG_System_Scenario_Rules
  VAR
    fbSystemScenarioArb : FB_System_Scenario_Arbitration;
    fbRuleEngine : FB_Rule_Engine;
    L_i : INT;
    L_Scenario_Req_Operator : E_SCENARIO_TYPE;
    L_Scenario_Req_Gateway : E_SCENARIO_TYPE;
    L_Scenario_Req_Rule : E_SCENARIO_TYPE;
    L_Scenario_Req_Final : E_SCENARIO_TYPE;
    L_Scenario_Intent : E_SCENARIO_TYPE;
    L_Scenario_Source : E_SCENARIO_SOURCE;
    L_Motion_16 : ARRAY[1..16] OF BOOL;
  END_VAR

            // adapt motion sensors (32 → 16)
FOR L_i := 1 TO 16 DO
    L_Motion_16[L_i] := GVL_STATE.G_Motion_Sensors[L_i];
END_FOR;

IF GVL_STATE.G_System_Mode = E_System_Operating_Mode.MODE_NORMAL THEN
    L_Scenario_Req_Operator := GVL_COMMAND.G_Scenario_Request_Operator;
ELSE
    L_Scenario_Req_Operator := E_SCENARIO_TYPE.SCENARIO_NONE;
END_IF;

L_Scenario_Req_Gateway := GVL_INTENT_USER.I_Scenario_Request;
L_Scenario_Req_Rule := E_SCENARIO_TYPE.SCENARIO_NONE;

fbRuleEngine(
    VI_System_Time_MS := GVL_TIME_SERVICE.G_Now_MS,
    VI_IsActivePLC := GVL_STATUS.G_Is_Active_PLC,
    VI_Security_Armed := GVL_ALARM.G_Security_Armed,
    VI_Current_Time := GVL_TIME_SERVICE.G_Current_TOD,
    VI_Day_Of_Week := GVL_TIME_SERVICE.G_Day_Of_Week,
    VI_Rules := GVL_CONFIG.G_HMI_User_Rules,
    VI_Indoor_Temps := GVL_STATE.G_Room_Temps,
    VI_Floor_Temps := GVL_STATE.G_Floor_Temps,
    VI_Humidities := GVL_STATE.G_Room_Hum,
    VI_CO2_Levels := GVL_STATE.G_Room_CO2,
    VI_Motion_Sensors := L_Motion_16,
    VI_Door_Sensors := GVL_STATE.G_Door_Sensors,
    VI_Window_Sensors := GVL_STATE.G_Window_Sensors,
    VI_Water_Sensors := GVL_STATE.G_Water_Sensors,
    VI_Smoke_Sensors := GVL_STATE.G_Smoke_Sensors,
    VI_Methane_Sensors := GVL_STATE.G_Methane_Sensors,
    VI_CO_Sensors := GVL_STATE.G_CO_Sensors,
    VO_Actions => GVL_STATE.G_Rule_Actions
);

FOR L_i := 1 TO GVL_CONSTANTS.C_MAX_RULES DO
    IF GVL_STATE.G_Rule_Actions[L_i].Active AND GVL_STATE.G_Rule_Actions[L_i].Action_Type = E_Rule_Action_Type.ACTION_ACTIVATE_SCENARIO THEN
        L_Scenario_Req_Rule := TO_BYTE(GVL_STATE.G_Rule_Actions[L_i].Value);
    END_IF;
END_FOR;

fbSystemScenarioArb(
    VI_System_Time_MS := GVL_TIME_SERVICE.G_Now_MS,
    VI_IsActivePLC := GVL_STATUS.G_Is_Active_PLC,
    VI_System_Mode := GVL_STATE.G_System_Mode,
    VI_Security_Armed := GVL_ALARM.G_Security_Armed,
    VIO_Scenario_Req_Operator := L_Scenario_Req_Operator,
    VIO_Scenario_Req_Gateway := L_Scenario_Req_Gateway,
    VIO_Scenario_Req_Rule := L_Scenario_Req_Rule,
    VIO_Scenario_Req_Final := L_Scenario_Req_Final,
    VIO_Scenario_Intent := L_Scenario_Intent,
    VIO_Scenario_Source := L_Scenario_Source
);
          
END_PROGRAM

PROGRAM PRG_Observability_Authority_Governor
  VAR
    L_Now_MS : UDINT;
    L_Observability_Valid : BOOL := TRUE;
  END_VAR

            L_Now_MS := GVL_STATUS.G_System_Time_MS;
L_Observability_Valid := TRUE;

// Fail-safe defaults.
GVL_OBSERVABILITY_AUTHORITY_FABRIC.Observability_Authority_Valid := FALSE;
GVL_OBSERVABILITY_AUTHORITY_FABRIC.Observability_Quarantine_Active := TRUE;
GVL_OBSERVABILITY_AUTHORITY_FABRIC.Observability_Publication_Allowed := FALSE;

GVL_OBSERVABILITY_AUTHORITY_FABRIC.HMI_Authority_Coherent := FALSE;
GVL_OBSERVABILITY_AUTHORITY_FABRIC.Diagnostics_Authority_Coherent := FALSE;
GVL_OBSERVABILITY_AUTHORITY_FABRIC.Blackbox_Authority_Coherent := FALSE;
GVL_OBSERVABILITY_AUTHORITY_FABRIC.Trend_Authority_Coherent := FALSE;
GVL_OBSERVABILITY_AUTHORITY_FABRIC.Alarm_Authority_Coherent := FALSE;

// Revocation blocks authoritative observability.
IF GVL_AUTHORITY_REVOCATION.Authority_Revocation_Active THEN
    L_Observability_Valid := FALSE;
END_IF;

// Restoration must be fully completed.
IF L_Observability_Valid
AND NOT GVL_AUTHORITY_RESTORATION.Authority_Restoration_Completed THEN
    L_Observability_Valid := FALSE;
END_IF;

// Physical authority epoch coherence required.
IF L_Observability_Valid
AND NOT GVL_PHYSICAL_AUTHORITY_EPOCH.Physical_Authority_Epoch_Valid THEN
    L_Observability_Valid := FALSE;
END_IF;

// Authority lineage continuity required.
IF L_Observability_Valid
AND NOT GVL_AUTHORITY_LINEAGE.Authority_Lineage_Valid THEN
    L_Observability_Valid := FALSE;
END_IF;

IF L_Observability_Valid THEN
    GVL_OBSERVABILITY_AUTHORITY_FABRIC.Observability_Authority_Valid := TRUE;
    GVL_OBSERVABILITY_AUTHORITY_FABRIC.Observability_Quarantine_Active := FALSE;
    GVL_OBSERVABILITY_AUTHORITY_FABRIC.Observability_Publication_Allowed := TRUE;

    GVL_OBSERVABILITY_AUTHORITY_FABRIC.HMI_Authority_Coherent := TRUE;
    GVL_OBSERVABILITY_AUTHORITY_FABRIC.Diagnostics_Authority_Coherent := TRUE;
    GVL_OBSERVABILITY_AUTHORITY_FABRIC.Blackbox_Authority_Coherent := TRUE;
    GVL_OBSERVABILITY_AUTHORITY_FABRIC.Trend_Authority_Coherent := TRUE;
    GVL_OBSERVABILITY_AUTHORITY_FABRIC.Alarm_Authority_Coherent := TRUE;

    GVL_OBSERVABILITY_AUTHORITY_FABRIC.Observability_Epoch :=
        GVL_PHYSICAL_AUTHORITY_EPOCH.Physical_Authority_Epoch;

    GVL_OBSERVABILITY_AUTHORITY_FABRIC.Observability_Epoch_Coherent := TRUE;

    GVL_OBSERVABILITY_AUTHORITY_FABRIC.Observability_Last_Update_MS :=
        L_Now_MS;

    GVL_OBSERVABILITY_AUTHORITY_FABRIC.Observability_Lease_Expired := FALSE;
ELSE
    GVL_OBSERVABILITY_AUTHORITY_FABRIC.Observability_Authority_Valid := FALSE;
    GVL_OBSERVABILITY_AUTHORITY_FABRIC.Observability_Quarantine_Active := TRUE;
    GVL_OBSERVABILITY_AUTHORITY_FABRIC.Observability_Publication_Allowed := FALSE;

    GVL_OBSERVABILITY_AUTHORITY_FABRIC.Observability_Lease_Expired := TRUE;

    GVL_OBSERVABILITY_AUTHORITY_FABRIC.Observability_Invalidation_Count :=
        GVL_OBSERVABILITY_AUTHORITY_FABRIC.Observability_Invalidation_Count + 1;
END_IF;
          
END_PROGRAM

PROGRAM PRG_Command_Verifier
  VAR
    L_i : INT;
    L_Mismatch_Count : INT := 0;
    L_Runtime_Error : BOOL := FALSE;
    L_Runtime_Error_Code : UDINT := 0;
    L_Runtime_Error_Text : STRING(160) := '';
    L_Now_MS : UDINT;
    L_Prev_Runtime_Error : BOOL;
    L_Any_Manifold_Pump_On : BOOL;
    fbLog : FB_LogEvent;
  END_VAR

            L_Now_MS := GVL_STATUS.G_System_Time_MS;

// ===============================
// 1. COMMAND MISMATCH CHECK
// ===============================
L_Mismatch_Count := 0;

IF GVL_COMMAND.G_Gas_Valve_Close <> GVL_COMMAND_SHADOW.G_Gas_Valve_Close THEN L_Mismatch_Count := L_Mismatch_Count + 1; END_IF;
IF GVL_COMMAND.G_Boiler_Stop <> GVL_COMMAND_SHADOW.G_Boiler_Stop THEN L_Mismatch_Count := L_Mismatch_Count + 1; END_IF;
IF GVL_COMMAND.G_Vent_Stop <> GVL_COMMAND_SHADOW.G_Vent_Stop THEN L_Mismatch_Count := L_Mismatch_Count + 1; END_IF;
IF GVL_COMMAND.G_Supply_100_Req <> GVL_COMMAND_SHADOW.G_Supply_100_Req THEN L_Mismatch_Count := L_Mismatch_Count + 1; END_IF;
IF GVL_COMMAND.G_Supply_80_Req <> GVL_COMMAND_SHADOW.G_Supply_80_Req THEN L_Mismatch_Count := L_Mismatch_Count + 1; END_IF;
IF GVL_COMMAND.G_Vent_PV3_Boost <> GVL_COMMAND_SHADOW.G_Vent_PV3_Boost THEN L_Mismatch_Count := L_Mismatch_Count + 1; END_IF;
IF GVL_COMMAND.G_Close_Valve_35 <> GVL_COMMAND_SHADOW.G_Close_Valve_35 THEN L_Mismatch_Count := L_Mismatch_Count + 1; END_IF;
IF GVL_COMMAND.G_Close_Valve_36 <> GVL_COMMAND_SHADOW.G_Close_Valve_36 THEN L_Mismatch_Count := L_Mismatch_Count + 1; END_IF;
IF GVL_COMMAND.G_Lock_1_Open <> GVL_COMMAND_SHADOW.G_Lock_1_Open THEN L_Mismatch_Count := L_Mismatch_Count + 1; END_IF;
IF GVL_COMMAND.G_Lock_1_Close <> GVL_COMMAND_SHADOW.G_Lock_1_Close THEN L_Mismatch_Count := L_Mismatch_Count + 1; END_IF;
IF GVL_COMMAND.G_Lock_2_Open <> GVL_COMMAND_SHADOW.G_Lock_2_Open THEN L_Mismatch_Count := L_Mismatch_Count + 1; END_IF;
IF GVL_COMMAND.G_Lock_2_Close <> GVL_COMMAND_SHADOW.G_Lock_2_Close THEN L_Mismatch_Count := L_Mismatch_Count + 1; END_IF;
IF GVL_COMMAND.G_Gate_Open <> GVL_COMMAND_SHADOW.G_Gate_Open THEN L_Mismatch_Count := L_Mismatch_Count + 1; END_IF;
IF GVL_COMMAND.G_Wicket_Open <> GVL_COMMAND_SHADOW.G_Wicket_Open THEN L_Mismatch_Count := L_Mismatch_Count + 1; END_IF;

GVL_COMMAND_VERIFY.Command_Mismatch_Count := L_Mismatch_Count;
GVL_COMMAND_VERIFY.Command_Match_OK := (L_Mismatch_Count = 0);
GVL_COMMAND_VERIFY.Command_Mismatch_Active := (L_Mismatch_Count > 0);

// ===============================
// 2. RUNTIME SANITY CHECKS
// ===============================
L_Runtime_Error := FALSE;
L_Runtime_Error_Code := 0;
L_Runtime_Error_Text := '';
L_Any_Manifold_Pump_On := FALSE;

// PLC inactive: fail-safe outputs should be off/safe except alarm/gas close outputs.
IF (NOT L_Runtime_Error) AND (NOT GVL_STATUS.G_Is_Active_PLC) THEN
    FOR L_i := 1 TO GVL_CONSTANTS.C_MAX_HEATING_CIRCUITS DO
        IF GVL_IO.DO_Zone_Valves[L_i] THEN
            L_Runtime_Error := TRUE;
            L_Runtime_Error_Code := 10;
            L_Runtime_Error_Text := 'PLC inactive zone valve on';
        END_IF;
    END_FOR;
END_IF;

IF (NOT L_Runtime_Error) AND (NOT GVL_STATUS.G_Is_Active_PLC) THEN
    FOR L_i := 1 TO GVL_CONSTANTS.C_MAX_MANIFOLDS DO
        IF GVL_IO.DO_Manifold_Pumps[L_i] THEN
            L_Runtime_Error := TRUE;
            L_Runtime_Error_Code := 11;
            L_Runtime_Error_Text := 'PLC inactive pump on';
        END_IF;
    END_FOR;
END_IF;

// GAS: gas valve must be physically commanded closed.
IF (NOT L_Runtime_Error) AND (GVL_SAFETY_SHUTDOWN.G_Safety_Mode = GAS) AND (NOT GVL_IO.DO_Gas_Valve_Close) THEN
    L_Runtime_Error := TRUE;
    L_Runtime_Error_Code := 1;
    L_Runtime_Error_Text := 'Gas valve not closed';
END_IF;

// GAS: ventilation must not be forced fully off by the IO layer.
IF (NOT L_Runtime_Error) AND (GVL_SAFETY_SHUTDOWN.G_Safety_Mode = GAS) THEN
    IF (GVL_IO.AO_Supply_Fans[1] = 0) AND (GVL_IO.AO_Exhaust_Fans[1] = 0) THEN
        L_Runtime_Error := TRUE;
        L_Runtime_Error_Code := 3;
        L_Runtime_Error_Text := 'Gas ventilation inactive';
    END_IF;
END_IF;

// FIRE: all exhaust fans should be commanded above zero in smoke exhaust mode.
IF (NOT L_Runtime_Error) AND (GVL_SAFETY_SHUTDOWN.G_Safety_Mode = FIRE) THEN
    FOR L_i := 1 TO GVL_CONSTANTS.C_MAX_EXHAUST_FANS DO
        IF GVL_IO.AO_Exhaust_Fans[L_i] = 0 THEN
            L_Runtime_Error := TRUE;
            L_Runtime_Error_Code := 2;
            L_Runtime_Error_Text := 'Smoke exhaust not active';
        END_IF;
    END_FOR;
END_IF;

// FIRE: supply fans should be off in smoke exhaust mode.
IF (NOT L_Runtime_Error) AND (GVL_SAFETY_SHUTDOWN.G_Safety_Mode = FIRE) THEN
    FOR L_i := 1 TO GVL_CONSTANTS.C_MAX_SUPPLY_FANS DO
        IF GVL_IO.AO_Supply_Fans[L_i] <> 0 THEN
            L_Runtime_Error := TRUE;
            L_Runtime_Error_Code := 4;
            L_Runtime_Error_Text := 'Supply fan active in fire';
        END_IF;
    END_FOR;
END_IF;

// WATER_LEAK: valve close commands must reach physical outputs.
IF (NOT L_Runtime_Error) AND (GVL_SAFETY_SHUTDOWN.G_Safety_Mode = WATER_LEAK) THEN
    IF GVL_COMMAND_SHADOW.G_Close_Valve_35 AND (NOT GVL_IO.DO_Water_Valve_35_Close) THEN
        L_Runtime_Error := TRUE;
        L_Runtime_Error_Code := 5;
        L_Runtime_Error_Text := 'Water valve 35 not closed';
    ELSIF GVL_COMMAND_SHADOW.G_Close_Valve_36 AND (NOT GVL_IO.DO_Water_Valve_36_Close) THEN
        L_Runtime_Error := TRUE;
        L_Runtime_Error_Code := 6;
        L_Runtime_Error_Text := 'Water valve 36 not closed';
    END_IF;
END_IF;

// FREEZE: when freeze-risk is active, heating circulation should not be fully dead.
IF (NOT L_Runtime_Error) AND GVL_STATE.G_Safety_Freeze_Risk THEN
    FOR L_i := 1 TO GVL_CONSTANTS.C_MAX_MANIFOLDS DO
        IF GVL_IO.DO_Manifold_Pumps[L_i] THEN
            L_Any_Manifold_Pump_On := TRUE;
        END_IF;
    END_FOR;

    IF (NOT L_Any_Manifold_Pump_On) AND (NOT GVL_IO.DO_Backup_Circulation_Pump) THEN
        L_Runtime_Error := TRUE;
        L_Runtime_Error_Code := 7;
        L_Runtime_Error_Text := 'Freeze circulation inactive';
    END_IF;
END_IF;

// GAS+FREEZE: electric backup may be used for anti-freeze, but DHW heating must remain off.
IF (NOT L_Runtime_Error) AND GVL_STATE.G_Safety_Freeze_Risk AND GVL_COMMAND_SHADOW.G_Heating_Gas_Safety_Stop THEN
    IF GVL_IO.DO_DHW_Heating_Pump THEN
        L_Runtime_Error := TRUE;
        L_Runtime_Error_Code := 8;
        L_Runtime_Error_Text := 'DHW heating active during gas freeze';
    END_IF;
END_IF;

// Apply result
IF L_Runtime_Error THEN
    GVL_COMMAND_VERIFY.Runtime_Sanity_OK := FALSE;
    GVL_COMMAND_VERIFY.Runtime_Last_Error_Code := L_Runtime_Error_Code;
    GVL_COMMAND_VERIFY.Runtime_Last_Error_Text := L_Runtime_Error_Text;
    GVL_COMMAND_VERIFY.Runtime_Last_Error_Time_MS := L_Now_MS;

    IF NOT L_Prev_Runtime_Error THEN
        GVL_COMMAND_VERIFY.Runtime_Sanity_Error_Count := GVL_COMMAND_VERIFY.Runtime_Sanity_Error_Count + 1;
        fbLog(
            VI_Event_Type := 1001,
            VI_Timestamp := L_Now_MS,
            VI_Param1 := L_Runtime_Error_Code,
            VI_Param2 := GVL_COMMAND_VERIFY.Runtime_Sanity_Error_Count
        );
    END_IF;
ELSE
    GVL_COMMAND_VERIFY.Runtime_Sanity_OK := TRUE;
END_IF;

L_Prev_Runtime_Error := L_Runtime_Error;
          
END_PROGRAM

PROGRAM PRG_PLC_A

            // Вызов основной программы
PRG_System();
// >>> BULK_SYNC_ANCHOR: PRG_PLC_A <<<
          
END_PROGRAM

PROGRAM PRG_System_Init
  VAR
    L_i : INT;
    L_Init_Done : BOOL := FALSE;
    L_Active_Zones_Count : INT;
    L_Zone_Index : INT;
  END_VAR

            IF L_Init_Done THEN
    RETURN;
END_IF;

// ======================================================
// SYSTEM INIT VALIDATION
// ======================================================
// Performs one-shot base system configuration checks.
//
// This PRG may publish status text, but it must not mutate
// aggregated diagnostics fields directly. Diagnostics aggregate
// ownership is centralized in FB_System_Health_Orchestrator.
//
// Runtime operational command authority is owned by
// PRG_Command_Arbitration.
// ======================================================

L_Active_Zones_Count := GVL_SYSTEM_SIZE_CONFIG.G_Active_Heating_Circuits;

IF (L_Active_Zones_Count < 1) OR (L_Active_Zones_Count > GVL_CONSTANTS.C_MAX_HEATING_CIRCUITS) THEN
    GVL_STATUS.G_System_Mode_Text := 'CONFIG ERROR: invalid active heating circuits';
    L_Active_Zones_Count := GVL_CONSTANTS.C_MAX_HEATING_CIRCUITS;
END_IF;

FOR L_i := 1 TO L_Active_Zones_Count DO
    L_Zone_Index := GVL_CONFIG.G_Heating_Circuit_To_Zone[L_i];
    IF (L_Zone_Index < 1) OR (L_Zone_Index > GVL_CONSTANTS.C_MAX_ZONES) THEN
        GVL_STATUS.G_System_Mode_Text := CONCAT('CONFIG ERROR CIRCUIT ', INT_TO_STRING(L_i));
    END_IF;
END_FOR;

L_Init_Done := TRUE;

// >>> BULK_SYNC_ANCHOR: PRG_System_Init <<<
          
END_PROGRAM

PROGRAM PRG_Semantic_Execution_Control_Governor

            // SEMANTIC EXECUTION COLLAPSE PREVENTION
// DETERMINISTIC SEMANTIC SCHEDULING
// NON-INVASIVE / ADVISORY-FIRST

IF GVL_RUNTIME_BUDGET_ENFORCEMENT.Runtime_Budget_Pressure_Observed THEN
    GVL_SEMANTIC_EXECUTION_CONTROL.Diagnostics_Execution_Path := DEFERRED_PATH;
    GVL_SEMANTIC_EXECUTION_CONTROL.Trend_Analytics_Execution_Path := BACKGROUND_PATH;
END_IF;

IF GVL_CANONICAL_RUNTIME_FABRIC_REGISTRY.Governance_Depth_Limit_Reached THEN
    GVL_SEMANTIC_EXECUTION_CONTROL.Semantic_Chain_Depth_Limit_Reached := TRUE;
    GVL_SEMANTIC_EXECUTION_CONTROL.Semantic_Execution_Fragmentation_Risk := TRUE;
END_IF;

IF GVL_CANONICAL_RUNTIME_FABRIC_REGISTRY.Verification_Chaining_Limit_Reached THEN
    GVL_SEMANTIC_EXECUTION_CONTROL.Verification_Fanout_Limit_Reached := TRUE;
    GVL_SEMANTIC_EXECUTION_CONTROL.Semantic_Cascade_Amplification_Risk := TRUE;
END_IF;

IF GVL_CANONICAL_RUNTIME_FABRIC_REGISTRY.Observability_Amplification_Limit_Reached THEN
    GVL_SEMANTIC_EXECUTION_CONTROL.Observability_Fanout_Limit_Reached := TRUE;
END_IF;

IF GVL_SURVIVABILITY_INTELLIGENCE_FABRIC.Chronic_Degradation_Risk_Increasing THEN
    GVL_SEMANTIC_EXECUTION_CONTROL.Semantic_Complexity_Ceiling_Reached := TRUE;
    GVL_SEMANTIC_EXECUTION_CONTROL.Autonomous_Complexity_Ceiling_Enforced := TRUE;
END_IF;

// Critical execution paths remain immediate.
GVL_SEMANTIC_EXECUTION_CONTROL.Safety_Execution_Path := FAST_PATH;
GVL_SEMANTIC_EXECUTION_CONTROL.Physical_Verification_Path := FAST_PATH;
          
END_PROGRAM

PROGRAM PRG_Causal_Narrative_Engine

            // PASSIVE CAUSAL NARRATIVE ENGINE
// HUMAN-READABLE SEMANTIC PROJECTION

GVL_CAUSAL_NARRATIVE_FABRIC.Narrative_Causality_Coherent :=
    GVL_TEMPORAL_CAUSALITY_CLOSURE_FABRIC.Temporal_Causality_Coherent;

GVL_CAUSAL_NARRATIVE_FABRIC.Narrative_Runtime_Alignment_Valid :=
    GVL_RUNTIME_TRANSITION_SYSTEM.Runtime_Transition_Legal;

IF GVL_RUNTIME_TRANSITION_SYSTEM.Illegal_Runtime_Transition_Observed THEN
    GVL_CAUSAL_NARRATIVE_FABRIC.Runtime_Narrative_Available := TRUE;
    GVL_CAUSAL_NARRATIVE_FABRIC.Runtime_Narrative_Code :=
        'transition legality violation observed';
END_IF;

IF GVL_RUNTIME_TRANSITION_SYSTEM.Recovery_Without_Lineage_Observed THEN
    GVL_CAUSAL_NARRATIVE_FABRIC.Recovery_Narrative_Available := TRUE;
    GVL_CAUSAL_NARRATIVE_FABRIC.Recovery_Narrative_Code :=
        'recovery blocked by lineage instability';
END_IF;

IF GVL_RUNTIME_TRANSITION_SYSTEM.Unsafe_Trust_Escalation_Observed THEN
    GVL_CAUSAL_NARRATIVE_FABRIC.Authority_Narrative_Available := TRUE;
    GVL_CAUSAL_NARRATIVE_FABRIC.Authority_Narrative_Code :=
        'unsafe trust escalation detected';
END_IF;
          
END_PROGRAM

PROGRAM PRG_Heating_Policy_Manager
  VAR
    fbPolicyManager : FB_Heating_Policy_Manager;
    fbSchedule : FB_Heating_Schedule_Preheat;
    fbThermal : FB_Heating_Thermal_Model;
    fbPredictive : FB_Heating_Predictive_Controller;
    fbOptimizer : FB_Heating_Optimizer;
    fbTime : FB_Time_Service;
    L_i : INT;
    L_Room_Avg : REAL;
    L_Floor_Avg : REAL;
  END_VAR

            fbTime();
fbThermal();
fbPredictive();
fbOptimizer();

L_Room_Avg := 0.0;
L_Floor_Avg := 0.0;

FOR L_i := 1 TO GVL_CONSTANTS.C_MAX_ZONES DO
    L_Room_Avg := L_Room_Avg + GVL_STATE.G_Room_Temps[L_i];
    L_Floor_Avg := L_Floor_Avg + GVL_STATE.G_Floor_Temps[L_i];
END_FOR;

L_Room_Avg := L_Room_Avg / TO_REAL(GVL_CONSTANTS.C_MAX_ZONES);
L_Floor_Avg := L_Floor_Avg / TO_REAL(GVL_CONSTANTS.C_MAX_ZONES);

fbPolicyManager(
    VI_System_Time_MS := GVL_TIME_SERVICE.G_Now_MS,
    VI_System_Mode := GVL_STATE.G_System_Mode,
    VI_RootCause := GVL_STATE.G_Heating_RootCause,
    VI_RootConfidence := GVL_STATE.G_Heating_RootConfidence,
    VI_Min_Hold_MS := GVL_CONFIG.G_Policy_Min_Hold_MS,
    VI_Emergency_Stop := GVL_STATE.G_Safety_Emergency_Stop,
    VI_Gas_Safety := GVL_STATE.G_Safety_Gas_Latched,
    VI_Room_Temp_Avg := L_Room_Avg,
    VI_Floor_Temp_Avg := L_Floor_Avg,
    VI_Supply_Temp := GVL_STATE.G_Manifold_T_Supply[1],
    VI_Return_Temp := GVL_STATE.G_Manifold_T_Return[1],
    VI_Target_Temp := GVL_STATE.G_Target_Temperature,
    VI_Room_Temps := GVL_STATE.G_Room_Temps,
    VI_Floor_Temps := GVL_STATE.G_Floor_Temps
);

fbSchedule(
    VI_System_Time_MS := GVL_TIME_SERVICE.G_Now_MS,
    VI_Time_Of_Day_MS := GVL_TIME_SERVICE.G_Time_Of_Day_MS,
    VI_Day_Of_Week := GVL_TIME_SERVICE.G_Day_Of_Week,
    VI_Enable := TRUE
);

GVL_HEATING_POLICY.G_Policy_Mode := fbPolicyManager.VO_Policy_Mode;
GVL_HEATING_POLICY.G_Policy_Block_Heating_Request := fbPolicyManager.VO_Block_Heating;
GVL_HEATING_POLICY.G_Policy_Target_Adjustment := fbPolicyManager.VO_Target_Adjustment;
GVL_HEATING_POLICY.G_Policy_Priority_Multiplier := fbPolicyManager.VO_Priority_Multiplier;
GVL_HEATING_POLICY.G_Policy_Self_Tune_Active := fbPolicyManager.VO_Self_Tune_Active;
GVL_HEATING_POLICY.G_Policy_Self_Tune_Level := fbPolicyManager.VO_Self_Tune_Level;
GVL_HEATING_POLICY.G_Policy_Feedback_Stable := fbPolicyManager.VO_Feedback_Stable;
GVL_HEATING_POLICY.G_Policy_Feedback_Improving := fbPolicyManager.VO_Feedback_Improving;
GVL_HEATING_POLICY.G_Policy_Feedback_Quality := fbPolicyManager.VO_Feedback_Quality;
          
END_PROGRAM

PROGRAM PRG_Heating_Supervisory_Publication
  VAR
    fbCircuitExplainabilityAdapter : FB_Heating_Circuit_Explainability_Adapter;
    fbSourceStabilityObserver : FB_Heating_Source_Stability_Observer;
    fbSupervisoryEnrichment : FB_Heating_Runtime_Supervisory_Enrichment;
    fbSupervisoryPublicationAdapter : FB_Heating_Runtime_Supervisory_Publication_Adapter;
    L_i : INT;
    L_Cascade_Boiler_Count : UINT;
    L_OT_Command_Valid : BOOL;
    L_Runtime_Context : ST_Heating_Runtime_Context;
    L_Causality_Node : ST_Heating_Runtime_Causality_Node;
    L_Causality_Edge : ST_Heating_Runtime_Causality_Edge;
    L_Blackbox_Event : ST_Heating_Runtime_Blackbox_Event;
    L_Predictive_State : ST_Heating_Runtime_Predictive_State;
    L_Status_Code : UINT;
    L_Status_Text : STRING(128);
  END_VAR

            // ==============================================================================
// Heating supervisory publication orchestration
//
// Observation-only program.
// Runs after PRG_Heating has produced canonical runtime projection.
// Does not own runtime, outputs, commands or heating authority.
// ==============================================================================

// Compatibility publication from canonical runtime projection.
fbCircuitExplainabilityAdapter(
    VI_Enable := TRUE
);

// Per-circuit predictive source-stability observation from canonical projection.
fbSourceStabilityObserver(
    VI_Enable := TRUE,
    VI_System_Time_MS := GVL_STATUS.G_System_Time_MS
);

// Build a supervisory runtime context from the published runtime observation.
// This is an observation projection only. It does not mutate runtime execution.
L_Runtime_Context.Runtime_Enabled := GVL_Heating_Runtime_Observation.G_Runtime_Observation.Runtime_Active;
L_Runtime_Context.Runtime_Ready := GVL_Heating_Runtime_Observation.G_Runtime_Observation.Runtime_Ready;
L_Runtime_Context.Runtime_Fault := GVL_Heating_Runtime_Observation.G_Runtime_Observation.Runtime_Fault;
L_Runtime_Context.Current_Phase := GVL_Heating_Runtime_Observation.G_Runtime_Observation.Current_Phase;

L_Runtime_Context.Allow_DHW_Phase := TRUE;
L_Runtime_Context.Allow_Heating_Phase := TRUE;
L_Runtime_Context.Allow_Service_Gating_Phase := TRUE;
L_Runtime_Context.Allow_State_Publication_Phase := TRUE;
L_Runtime_Context.Allow_Diagnostics_Phase := TRUE;
L_Runtime_Context.Allow_Output_Projection_Phase := TRUE;

L_Runtime_Context.DHW_Executed := GVL_Heating_Runtime_Observation.G_Runtime_Observation.DHW_Heating_Active;
L_Runtime_Context.Heating_Executed := GVL_Heating_Runtime_Observation.G_Runtime_Observation.Heating_Runtime_Active;
L_Runtime_Context.Service_Gating_Executed := TRUE;
L_Runtime_Context.State_Publication_Executed := GVL_Heating_Runtime_Observation.G_Runtime_Observation.Heating_Output_Active;
L_Runtime_Context.Diagnostics_Executed := GVL_Heating_Runtime_Observation.G_Runtime_Observation.Diagnostics_Active;
L_Runtime_Context.Output_Projection_Executed := GVL_Heating_Runtime_Observation.G_Runtime_Observation.Output_Projection_Last_Observed;

L_Runtime_Context.DHW_Before_Heating_Valid := GVL_Heating_Runtime_Observation.G_Runtime_Observation.DHW_Before_Heating_Observed;
L_Runtime_Context.State_Publication_Before_Diagnostics_Valid := GVL_Heating_Runtime_Observation.G_Runtime_Observation.Diagnostics_After_Publication_Observed;
L_Runtime_Context.Output_Projection_Last_Valid := GVL_Heating_Runtime_Observation.G_Runtime_Observation.Output_Projection_Last_Observed;

L_Runtime_Context.Diagnostics_Isolation_Valid := GVL_Heating_Runtime_Observation.G_Runtime_Observation.Diagnostics_Ownership_Valid;
L_Runtime_Context.Explainability_Isolation_Valid := GVL_Heating_Runtime_Observation.G_Runtime_Observation.Explainability_Active;
L_Runtime_Context.Safety_Isolation_Valid := GVL_Heating_Runtime_Observation.G_Runtime_Observation.Safety_Ownership_Valid;
L_Runtime_Context.OpenTherm_Ownership_Valid := GVL_Heating_Runtime_Observation.G_Runtime_Observation.OpenTherm_Ownership_Valid;
L_Runtime_Context.Cascade_Ownership_Valid := GVL_Heating_Runtime_Observation.G_Runtime_Observation.Cascade_Ownership_Valid;

L_Runtime_Context.Runtime_Status_Code := GVL_Heating_Runtime_Observation.G_Runtime_Observation.Observation_Status_Code;
L_Runtime_Context.Runtime_Status_Text := GVL_Heating_Runtime_Observation.G_Runtime_Observation.Observation_Status_Text;

// Lightweight OT/cascade observation for supervisory enrichment context.
L_Cascade_Boiler_Count := 0;
L_OT_Command_Valid := TRUE;

FOR L_i := 1 TO GVL_CONSTANTS.C_MAX_BOILERS DO
    IF GVL_STATE.G_Boiler_OT_Online[L_i] THEN
        L_Cascade_Boiler_Count := L_Cascade_Boiler_Count + 1;
    END_IF;

    IF GVL_STATE.G_Boiler_OT_Enable[L_i] AND NOT GVL_STATE.G_Boiler_OT_Online[L_i] THEN
        L_OT_Command_Valid := FALSE;
    END_IF;
END_FOR;

// Supervisory enrichment owns timeline/event/reconstruction ingestion.
fbSupervisoryEnrichment(
    VI_Enable := TRUE,
    VI_System_Time_MS := GVL_STATUS.G_System_Time_MS,
    VI_Runtime_Context := L_Runtime_Context,
    VI_Phase_Event := GVL_Heating_Runtime_Explainability.G_Runtime_Phase_Event,
    VI_Anomaly := GVL_Heating_Runtime_Explainability.G_Runtime_Anomaly,
    VI_Cascade_Boiler_Count := L_Cascade_Boiler_Count,
    VI_OT_Command_Valid := L_OT_Command_Valid,
    VIO_Event_Buffer := GVL_Heating_Runtime_Explainability.G_Runtime_Event_Buffer,
    VIO_Execution_Timeline := GVL_Heating_Runtime_Explainability.G_Runtime_Execution_Timeline,
    VO_Causality_Node => L_Causality_Node,
    VO_Causality_Edge => L_Causality_Edge,
    VO_Blackbox_Event => L_Blackbox_Event,
    VO_Predictive_State => L_Predictive_State,
    VO_Status_Code => L_Status_Code,
    VO_Status_Text => L_Status_Text
);

// Canonical supervisory publication surface.
fbSupervisoryPublicationAdapter(
    VI_Enable := TRUE,
    VI_Predictive_State := L_Predictive_State,
    VI_Causality_Node := L_Causality_Node,
    VI_Causality_Edge := L_Causality_Edge,
    VI_Blackbox_Event := L_Blackbox_Event,
    VI_Anomaly := GVL_Heating_Runtime_Explainability.G_Runtime_Anomaly
);

// Keep existing runtime explainability GVL as a compatibility publication surface.
GVL_Heating_Runtime_Explainability.G_Runtime_Blackbox_Event := L_Blackbox_Event;
GVL_Heating_Runtime_Explainability.G_Runtime_Predictive_State := L_Predictive_State;
GVL_Heating_Runtime_Explainability.G_Runtime_Explainability_Publication_Valid := TRUE;
GVL_Heating_Runtime_Explainability.G_Runtime_Explainability_Status_Code := L_Status_Code;
GVL_Heating_Runtime_Explainability.G_Runtime_Explainability_Status_Text := L_Status_Text;

// >>> BULK_SYNC_ANCHOR: PRG_Heating_Supervisory_Publication <<<
          
END_PROGRAM

PROGRAM PRG_Environmental_Authority_Governor
  VAR
    L_Now_MS : UDINT;
    L_Environment_Valid : BOOL := TRUE;
    L_Error_Code : UDINT := 0;
    L_Error_Text : STRING(160) := '';
  END_VAR

            L_Now_MS := GVL_STATUS.G_System_Time_MS;
L_Environment_Valid := TRUE;
L_Error_Code := 0;
L_Error_Text := '';

// Fail-safe defaults.
GVL_ENVIRONMENTAL_AUTHORITY.Environmental_Authority_Valid := FALSE;
GVL_ENVIRONMENTAL_AUTHORITY.Environmental_Authority_Granted := FALSE;
GVL_ENVIRONMENTAL_AUTHORITY.Environmental_Quarantine_Active := TRUE;

GVL_ENVIRONMENTAL_AUTHORITY.External_Environment_Causally_Compatible := FALSE;
GVL_ENVIRONMENTAL_AUTHORITY.Utility_Environment_Stable := FALSE;
GVL_ENVIRONMENTAL_AUTHORITY.Hydraulic_Source_Stable := FALSE;
GVL_ENVIRONMENTAL_AUTHORITY.Thermal_Environment_Stable := FALSE;
GVL_ENVIRONMENTAL_AUTHORITY.Airflow_Environment_Stable := FALSE;

// Environmental authority requires temporal stability.
IF NOT GVL_TEMPORAL_STABILITY.Temporal_Stability_Granted THEN
    L_Environment_Valid := FALSE;
    L_Error_Code := 29000;
    L_Error_Text := 'Temporal stability authority not granted';
END_IF;

// Freeze propagation detection.
IF GVL_ENVIRONMENTAL_AUTHORITY.Freeze_Front_Propagation_Detected THEN
    L_Environment_Valid := FALSE;
    L_Error_Code := 29001;
    L_Error_Text := 'Freeze-front propagation detected';
END_IF;

// Utility instability propagation.
IF GVL_ENVIRONMENTAL_AUTHORITY.Utility_Instability_Propagation_Detected THEN
    L_Environment_Valid := FALSE;
    L_Error_Code := 29002;
    L_Error_Text := 'Utility instability propagation detected';
END_IF;

// Hydraulic collapse prediction.
IF GVL_ENVIRONMENTAL_AUTHORITY.External_Hydraulic_Collapse_Detected THEN
    L_Environment_Valid := FALSE;
    L_Error_Code := 29003;
    L_Error_Text := 'External hydraulic collapse detected';
END_IF;

// Airflow icing conditions.
IF GVL_ENVIRONMENTAL_AUTHORITY.Airflow_Icing_Condition_Detected THEN
    L_Environment_Valid := FALSE;
    L_Error_Code := 29004;
    L_Error_Text := 'Airflow icing condition detected';
END_IF;

// Environmental rebound race.
IF GVL_ENVIRONMENTAL_AUTHORITY.Environmental_Rebound_Race_Detected THEN
    L_Environment_Valid := FALSE;
    L_Error_Code := 29005;
    L_Error_Text := 'Environmental rebound race detected';
END_IF;

// External environment validation.
IF L_Environment_Valid
AND NOT GVL_ENVIRONMENTAL_AUTHORITY.Mains_Quality_Valid THEN
    L_Environment_Valid := FALSE;
    L_Error_Code := 29010;
    L_Error_Text := 'Mains quality invalid';
END_IF;

IF L_Environment_Valid
AND NOT GVL_ENVIRONMENTAL_AUTHORITY.Supply_Water_Available THEN
    L_Environment_Valid := FALSE;
    L_Error_Code := 29011;
    L_Error_Text := 'Supply water unavailable';
END_IF;

IF L_Environment_Valid
AND NOT GVL_ENVIRONMENTAL_AUTHORITY.Outdoor_Airflow_Valid THEN
    L_Environment_Valid := FALSE;
    L_Error_Code := 29012;
    L_Error_Text := 'Outdoor airflow invalid';
END_IF;

IF L_Environment_Valid
AND NOT GVL_ENVIRONMENTAL_AUTHORITY.Freeze_Protection_Valid THEN
    L_Environment_Valid := FALSE;
    L_Error_Code := 29013;
    L_Error_Text := 'Freeze protection invalid';
END_IF;

IF L_Environment_Valid THEN
    GVL_ENVIRONMENTAL_AUTHORITY.Environmental_Authority_Valid := TRUE;
    GVL_ENVIRONMENTAL_AUTHORITY.Environmental_Authority_Granted := TRUE;
    GVL_ENVIRONMENTAL_AUTHORITY.Environmental_Quarantine_Active := FALSE;

    GVL_ENVIRONMENTAL_AUTHORITY.External_Environment_Causally_Compatible := TRUE;
    GVL_ENVIRONMENTAL_AUTHORITY.Utility_Environment_Stable := TRUE;
    GVL_ENVIRONMENTAL_AUTHORITY.Hydraulic_Source_Stable := TRUE;
    GVL_ENVIRONMENTAL_AUTHORITY.Thermal_Environment_Stable := TRUE;
    GVL_ENVIRONMENTAL_AUTHORITY.Airflow_Environment_Stable := TRUE;

    GVL_ENVIRONMENTAL_AUTHORITY.Environmental_Authority_Epoch :=
        GVL_TEMPORAL_STABILITY.Temporal_Stability_Epoch;

    GVL_ENVIRONMENTAL_AUTHORITY.Environmental_Authority_Epoch_Coherent := TRUE;

    GVL_ENVIRONMENTAL_AUTHORITY.Environmental_Last_Update_MS :=
        L_Now_MS;

    GVL_ENVIRONMENTAL_AUTHORITY.Environmental_Lease_Expired := FALSE;

    GVL_ENVIRONMENTAL_AUTHORITY.Environmental_Last_Error_Code := 0;
    GVL_ENVIRONMENTAL_AUTHORITY.Environmental_Last_Error_Text := '';
ELSE
    GVL_ENVIRONMENTAL_AUTHORITY.Environmental_Authority_Valid := FALSE;
    GVL_ENVIRONMENTAL_AUTHORITY.Environmental_Authority_Granted := FALSE;
    GVL_ENVIRONMENTAL_AUTHORITY.Environmental_Quarantine_Active := TRUE;

    GVL_ENVIRONMENTAL_AUTHORITY.Environmental_Lease_Expired := TRUE;

    GVL_ENVIRONMENTAL_AUTHORITY.Environmental_Last_Error_Code :=
        L_Error_Code;

    GVL_ENVIRONMENTAL_AUTHORITY.Environmental_Last_Error_Text :=
        L_Error_Text;

    GVL_ENVIRONMENTAL_AUTHORITY.Environmental_Invalidation_Count :=
        GVL_ENVIRONMENTAL_AUTHORITY.Environmental_Invalidation_Count + 1;
END_IF;
          
END_PROGRAM

